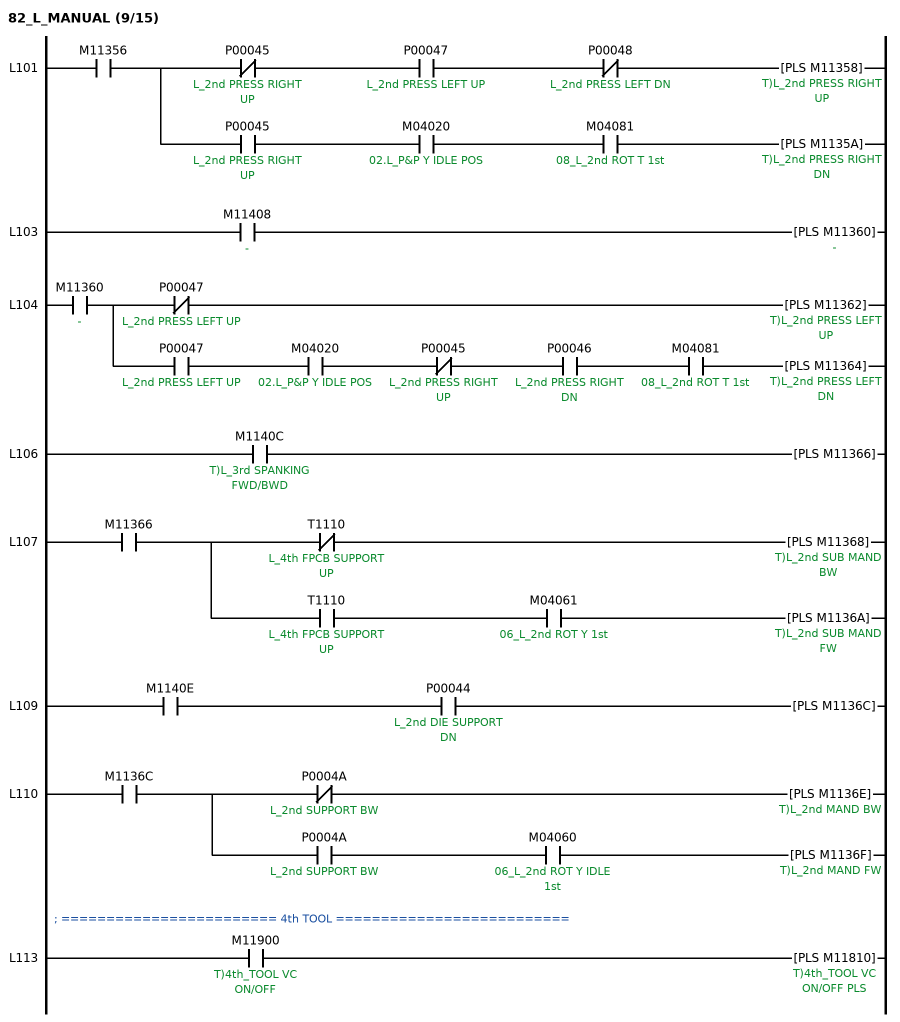
[picture p336: 82_L_MANUAL rungs L101-L113]
; L101
LOAD      M11356
MPUSH
AND NOT   P00045	// L_2nd PRESS RIGHT UP
AND       P00047	// L_2nd PRESS LEFT UP
AND NOT   P00048	// L_2nd PRESS LEFT DN
OUTP      M11358	// T)L_2nd PRESS RIGHT UP
MPOP
AND       P00045	// L_2nd PRESS RIGHT UP
AND       M04020	// 02.L_P&P Y IDLE POS
AND       M04081	// 08_L_2nd ROT T 1st
OUTP      M1135A	// T)L_2nd PRESS RIGHT DN
; L103
LOAD      M11408	// -
OUTP      M11360	// -
; L104
LOAD      M11360	// -
MPUSH
AND NOT   P00047	// L_2nd PRESS LEFT UP
OUTP      M11362	// T)L_2nd PRESS LEFT UP
MPOP
AND       P00047	// L_2nd PRESS LEFT UP
AND       M04020	// 02.L_P&P Y IDLE POS
AND NOT   P00045	// L_2nd PRESS RIGHT UP
AND       P00046	// L_2nd PRESS RIGHT DN
AND       M04081	// 08_L_2nd ROT T 1st
OUTP      M11364	// T)L_2nd PRESS LEFT DN
; L106
LOAD      M1140C	// T)L_3rd SPANKING FWD/BWD
OUTP      M11366
; L107
LOAD      M11366
MPUSH
AND NOT   T1110	// L_4th FPCB SUPPORT UP
OUTP      M11368	// T)L_2nd SUB MAND BW
MPOP
AND       T1110	// L_4th FPCB SUPPORT UP
AND       M04061	// 06_L_2nd ROT Y 1st
OUTP      M1136A	// T)L_2nd SUB MAND FW
; L109
LOAD      M1140E
AND       P00044	// L_2nd DIE SUPPORT DN
OUTP      M1136C
; L110
LOAD      M1136C
MPUSH
AND NOT   P0004A	// L_2nd SUPPORT BW
OUTP      M1136E	// T)L_2nd MAND BW
MPOP
AND       P0004A	// L_2nd SUPPORT BW
AND       M04060	// 06_L_2nd ROT Y IDLE 1st
OUTP      M1136F	// T)L_2nd MAND FW
// ======================== 4th TOOL ==========================
; L113
LOAD      M11900	// T)4th_TOOL VC ON/OFF
OUTP      M11810	// T)4th_TOOL VC ON/OFF PLS

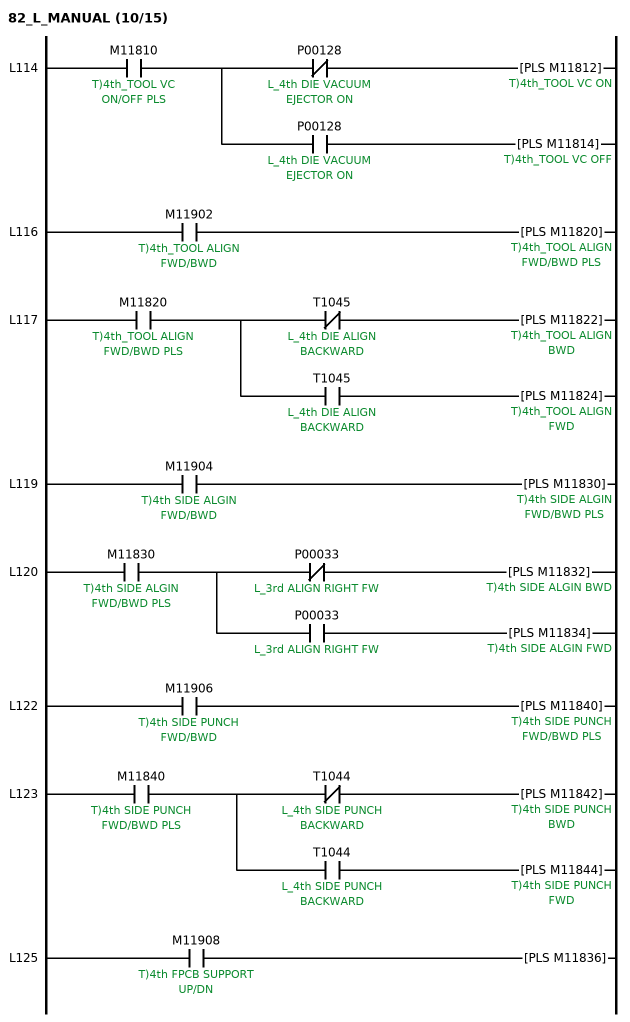
; L114
LOAD      M11810	// T)4th_TOOL VC ON/OFF PLS
MPUSH
AND NOT   P00128	// L_4th DIE VACUUM EJECTOR ON
OUTP      M11812	// T)4th_TOOL VC ON
MPOP
AND       P00128	// L_4th DIE VACUUM EJECTOR ON
OUTP      M11814	// T)4th_TOOL VC OFF
; L116
LOAD      M11902	// T)4th_TOOL ALIGN FWD/BWD
OUTP      M11820	// T)4th_TOOL ALIGN FWD/BWD PLS
; L117
LOAD      M11820	// T)4th_TOOL ALIGN FWD/BWD PLS
MPUSH
AND NOT   T1045	// L_4th DIE ALIGN BACKWARD
OUTP      M11822	// T)4th_TOOL ALIGN BWD
MPOP
AND       T1045	// L_4th DIE ALIGN BACKWARD
OUTP      M11824	// T)4th_TOOL ALIGN FWD
; L119
LOAD      M11904	// T)4th SIDE ALGIN FWD/BWD
OUTP      M11830	// T)4th SIDE ALGIN FWD/BWD PLS
; L120
LOAD      M11830	// T)4th SIDE ALGIN FWD/BWD PLS
MPUSH
AND NOT   P00033	// L_3rd ALIGN RIGHT FW
OUTP      M11832	// T)4th SIDE ALGIN BWD
MPOP
AND       P00033	// L_3rd ALIGN RIGHT FW
OUTP      M11834	// T)4th SIDE ALGIN FWD
; L122
LOAD      M11906	// T)4th SIDE PUNCH FWD/BWD
OUTP      M11840	// T)4th SIDE PUNCH FWD/BWD PLS
; L123
LOAD      M11840	// T)4th SIDE PUNCH FWD/BWD PLS
MPUSH
AND NOT   T1044	// L_4th SIDE PUNCH BACKWARD
OUTP      M11842	// T)4th SIDE PUNCH BWD
MPOP
AND       T1044	// L_4th SIDE PUNCH BACKWARD
OUTP      M11844	// T)4th SIDE PUNCH FWD
; L125
LOAD      M11908	// T)4th FPCB SUPPORT UP/DN
OUTP      M11836

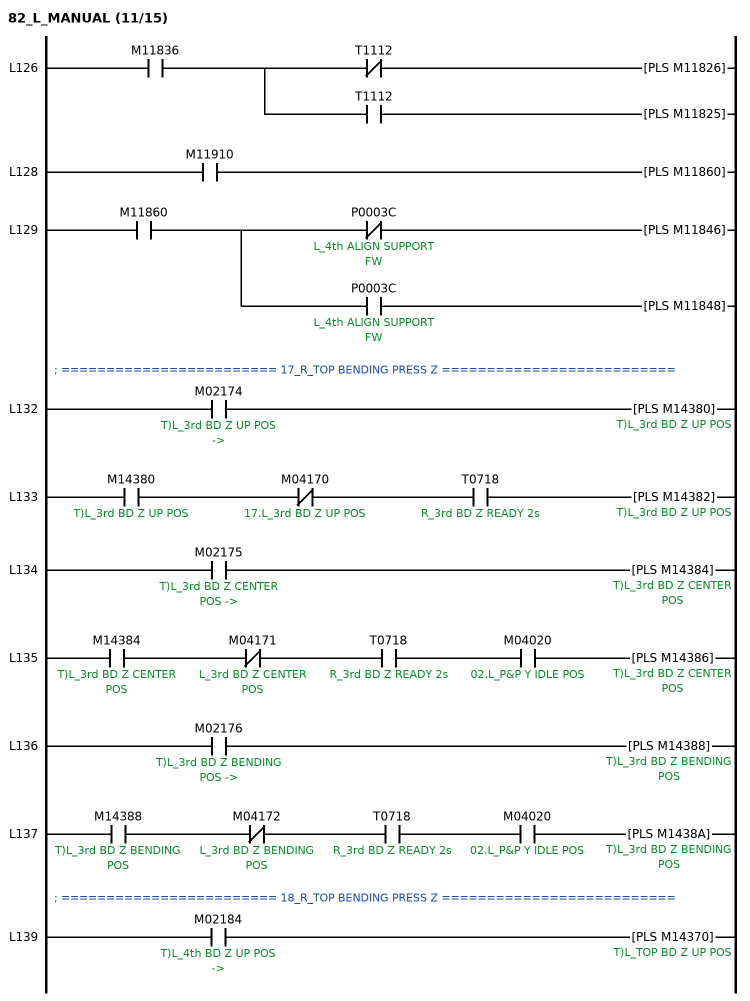
; L126
LOAD      M11836
MPUSH
AND NOT   T1112
OUTP      M11826
MPOP
AND       T1112
OUTP      M11825
; L128
LOAD      M11910
OUTP      M11860
; L129
LOAD      M11860
MPUSH
AND NOT   P0003C	// L_4th ALIGN SUPPORT FW
OUTP      M11846
MPOP
AND       P0003C	// L_4th ALIGN SUPPORT FW
OUTP      M11848
// ======================== 17_R_TOP BENDING PRESS Z ==========================
; L132
LOAD      M02174	// T)L_3rd BD Z UP POS ->
OUTP      M14380	// T)L_3rd BD Z UP POS
; L133
LOAD      M14380	// T)L_3rd BD Z UP POS
AND NOT   M04170	// 17.L_3rd BD Z UP POS
AND       T0718	// R_3rd BD Z READY 2s
OUTP      M14382	// T)L_3rd BD Z UP POS
; L134
LOAD      M02175	// T)L_3rd BD Z CENTER POS ->
OUTP      M14384	// T)L_3rd BD Z CENTER POS
; L135
LOAD      M14384	// T)L_3rd BD Z CENTER POS
AND NOT   M04171	// L_3rd BD Z CENTER POS
AND       T0718	// R_3rd BD Z READY 2s
AND       M04020	// 02.L_P&P Y IDLE POS
OUTP      M14386	// T)L_3rd BD Z CENTER POS
; L136
LOAD      M02176	// T)L_3rd BD Z BENDING POS ->
OUTP      M14388	// T)L_3rd BD Z BENDING POS
; L137
LOAD      M14388	// T)L_3rd BD Z BENDING POS
AND NOT   M04172	// L_3rd BD Z BENDING POS
AND       T0718	// R_3rd BD Z READY 2s
AND       M04020	// 02.L_P&P Y IDLE POS
OUTP      M1438A	// T)L_3rd BD Z BENDING POS
// ======================== 18_R_TOP BENDING PRESS Z ==========================
; L139
LOAD      M02184	// T)L_4th BD Z UP POS ->
OUTP      M14370	// T)L_TOP BD Z UP POS

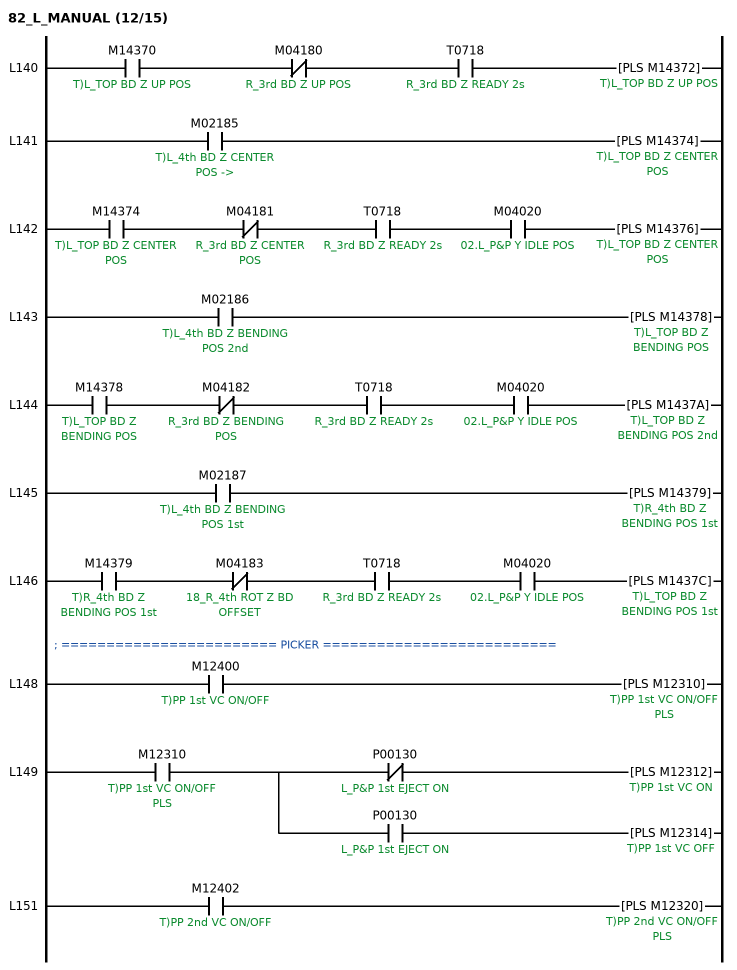
; L140
LOAD      M14370	// T)L_TOP BD Z UP POS
AND NOT   M04180	// R_3rd BD Z UP POS
AND       T0718	// R_3rd BD Z READY 2s
OUTP      M14372	// T)L_TOP BD Z UP POS
; L141
LOAD      M02185	// T)L_4th BD Z CENTER POS ->
OUTP      M14374	// T)L_TOP BD Z CENTER POS
; L142
LOAD      M14374	// T)L_TOP BD Z CENTER POS
AND NOT   M04181	// R_3rd BD Z CENTER POS
AND       T0718	// R_3rd BD Z READY 2s
AND       M04020	// 02.L_P&P Y IDLE POS
OUTP      M14376	// T)L_TOP BD Z CENTER POS
; L143
LOAD      M02186	// T)L_4th BD Z BENDING POS 2nd
OUTP      M14378	// T)L_TOP BD Z BENDING POS
; L144
LOAD      M14378	// T)L_TOP BD Z BENDING POS
AND NOT   M04182	// R_3rd BD Z BENDING POS
AND       T0718	// R_3rd BD Z READY 2s
AND       M04020	// 02.L_P&P Y IDLE POS
OUTP      M1437A	// T)L_TOP BD Z BENDING POS 2nd
; L145
LOAD      M02187	// T)L_4th BD Z BENDING POS 1st
OUTP      M14379	// T)R_4th BD Z BENDING POS 1st
; L146
LOAD      M14379	// T)R_4th BD Z BENDING POS 1st
AND NOT   M04183	// 18_R_4th ROT Z BD OFFSET
AND       T0718	// R_3rd BD Z READY 2s
AND       M04020	// 02.L_P&P Y IDLE POS
OUTP      M1437C	// T)L_TOP BD Z BENDING POS 1st
// ======================== PICKER ==========================
; L148
LOAD      M12400	// T)PP 1st VC ON/OFF
OUTP      M12310	// T)PP 1st VC ON/OFF PLS
; L149
LOAD      M12310	// T)PP 1st VC ON/OFF PLS
MPUSH
AND NOT   P00130	// L_P&P 1st EJECT ON
OUTP      M12312	// T)PP 1st VC ON
MPOP
AND       P00130	// L_P&P 1st EJECT ON
OUTP      M12314	// T)PP 1st VC OFF
; L151
LOAD      M12402	// T)PP 2nd VC ON/OFF
OUTP      M12320	// T)PP 2nd VC ON/OFF PLS

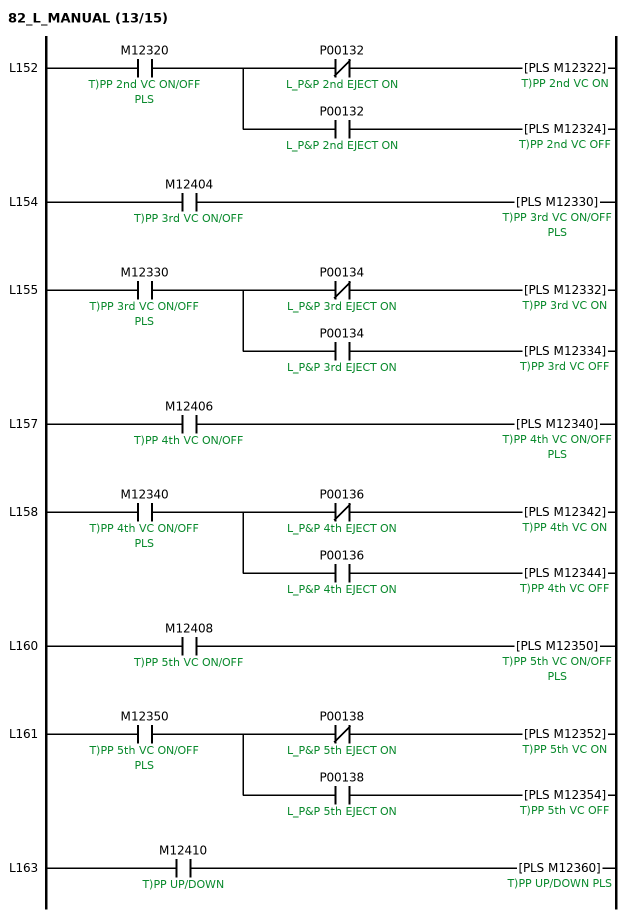
; L152
LOAD      M12320	// T)PP 2nd VC ON/OFF PLS
MPUSH
AND NOT   P00132	// L_P&P 2nd EJECT ON
OUTP      M12322	// T)PP 2nd VC ON
MPOP
AND       P00132	// L_P&P 2nd EJECT ON
OUTP      M12324	// T)PP 2nd VC OFF
; L154
LOAD      M12404	// T)PP 3rd VC ON/OFF
OUTP      M12330	// T)PP 3rd VC ON/OFF PLS
; L155
LOAD      M12330	// T)PP 3rd VC ON/OFF PLS
MPUSH
AND NOT   P00134	// L_P&P 3rd EJECT ON
OUTP      M12332	// T)PP 3rd VC ON
MPOP
AND       P00134	// L_P&P 3rd EJECT ON
OUTP      M12334	// T)PP 3rd VC OFF
; L157
LOAD      M12406	// T)PP 4th VC ON/OFF
OUTP      M12340	// T)PP 4th VC ON/OFF PLS
; L158
LOAD      M12340	// T)PP 4th VC ON/OFF PLS
MPUSH
AND NOT   P00136	// L_P&P 4th EJECT ON
OUTP      M12342	// T)PP 4th VC ON
MPOP
AND       P00136	// L_P&P 4th EJECT ON
OUTP      M12344	// T)PP 4th VC OFF
; L160
LOAD      M12408	// T)PP 5th VC ON/OFF
OUTP      M12350	// T)PP 5th VC ON/OFF PLS
; L161
LOAD      M12350	// T)PP 5th VC ON/OFF PLS
MPUSH
AND NOT   P00138	// L_P&P 5th EJECT ON
OUTP      M12352	// T)PP 5th VC ON
MPOP
AND       P00138	// L_P&P 5th EJECT ON
OUTP      M12354	// T)PP 5th VC OFF
; L163
LOAD      M12410	// T)PP UP/DOWN
OUTP      M12360	// T)PP UP/DOWN PLS

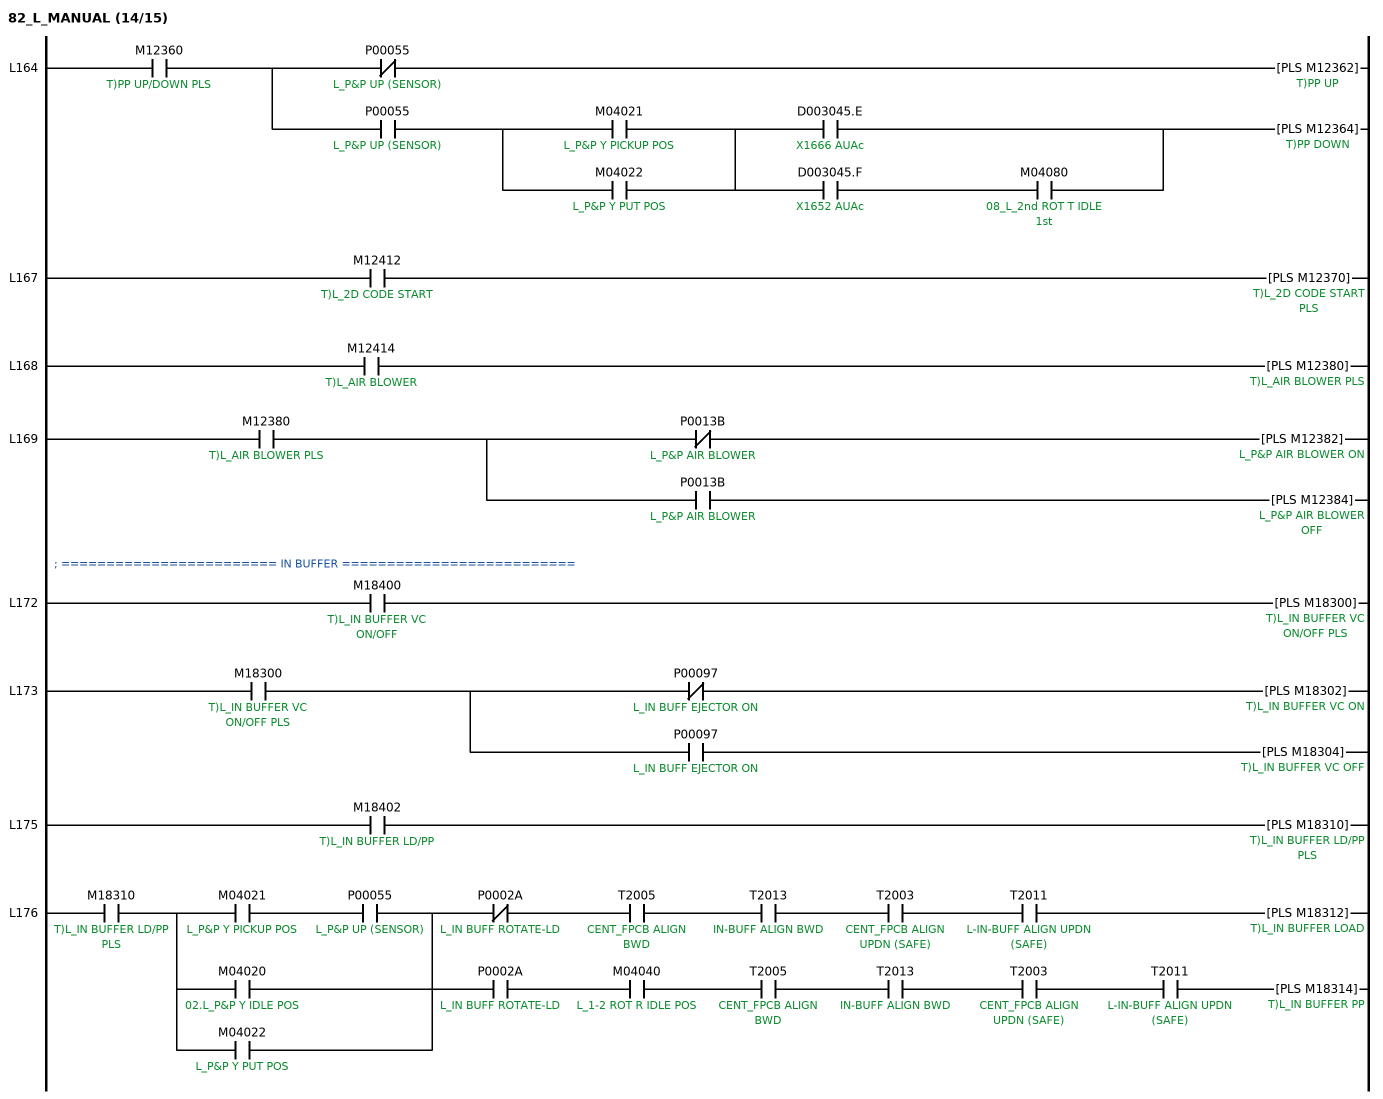
; L164
LOAD      M12360	// T)PP UP/DOWN PLS
MPUSH
AND NOT   P00055	// L_P&P UP (SENSOR)
OUTP      M12362	// T)PP UP
MPOP
AND       P00055	// L_P&P UP (SENSOR)
LOAD      M04021	// L_P&P Y PICKUP POS
OR        M04022	// L_P&P Y PUT POS
AND LOAD
LOAD      D003045.E	// X1666 AUAc
LOAD      D003045.F	// X1652 AUAc
AND       M04080	// 08_L_2nd ROT T IDLE 1st
OR LOAD
AND LOAD
OUTP      M12364	// T)PP DOWN
; L167
LOAD      M12412	// T)L_2D CODE START
OUTP      M12370	// T)L_2D CODE START PLS
; L168
LOAD      M12414	// T)L_AIR BLOWER
OUTP      M12380	// T)L_AIR BLOWER PLS
; L169
LOAD      M12380	// T)L_AIR BLOWER PLS
MPUSH
AND NOT   P0013B	// L_P&P AIR BLOWER
OUTP      M12382	// L_P&P AIR BLOWER ON
MPOP
AND       P0013B	// L_P&P AIR BLOWER
OUTP      M12384	// L_P&P AIR BLOWER OFF
// ======================== IN BUFFER ==========================
; L172
LOAD      M18400	// T)L_IN BUFFER VC ON/OFF
OUTP      M18300	// T)L_IN BUFFER VC ON/OFF PLS
; L173
LOAD      M18300	// T)L_IN BUFFER VC ON/OFF PLS
MPUSH
AND NOT   P00097	// L_IN BUFF EJECTOR ON
OUTP      M18302	// T)L_IN BUFFER VC ON
MPOP
AND       P00097	// L_IN BUFF EJECTOR ON
OUTP      M18304	// T)L_IN BUFFER VC OFF
; L175
LOAD      M18402	// T)L_IN BUFFER LD/PP
OUTP      M18310	// T)L_IN BUFFER LD/PP PLS
; L176
LOAD      M18310	// T)L_IN BUFFER LD/PP PLS
LOAD      M04021	// L_P&P Y PICKUP POS
AND       P00055	// L_P&P UP (SENSOR)
OR        M04020	// 02.L_P&P Y IDLE POS
OR        M04022	// L_P&P Y PUT POS
AND LOAD
MPUSH
AND NOT   P0002A	// L_IN BUFF ROTATE-LD
AND       T2005	// CENT_FPCB ALIGN BWD
AND       T2013	// IN-BUFF ALIGN BWD
AND       T2003	// CENT_FPCB ALIGN UPDN (SAFE)
AND       T2011	// L-IN-BUFF ALIGN UPDN (SAFE)
OUTP      M18312	// T)L_IN BUFFER LOAD
MPOP
AND       P0002A	// L_IN BUFF ROTATE-LD
AND       M04040	// L_1-2 ROT R IDLE POS
AND       T2005	// CENT_FPCB ALIGN BWD
AND       T2013	// IN-BUFF ALIGN BWD
AND       T2003	// CENT_FPCB ALIGN UPDN (SAFE)
AND       T2011	// L-IN-BUFF ALIGN UPDN (SAFE)
OUTP      M18314	// T)L_IN BUFFER PP

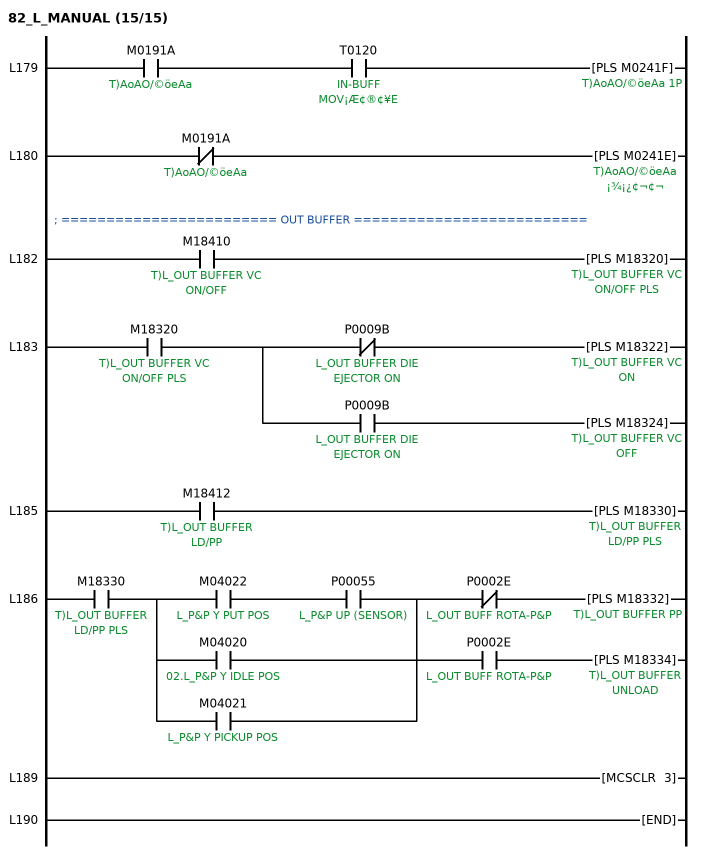
; L179
LOAD      M0191A	// T)AoAO/©öeAa
AND       T0120	// IN-BUFF MOV¡Æ¢®¢¥E
OUTP      M0241F	// T)AoAO/©öeAa 1P
; L180
LOAD NOT  M0191A	// T)AoAO/©öeAa
OUTP      M0241E	// T)AoAO/©öeAa ¡¾¡¿¢¬¢¬
// ======================== OUT BUFFER ==========================
; L182
LOAD      M18410	// T)L_OUT BUFFER VC ON/OFF
OUTP      M18320	// T)L_OUT BUFFER VC ON/OFF PLS
; L183
LOAD      M18320	// T)L_OUT BUFFER VC ON/OFF PLS
MPUSH
AND NOT   P0009B	// L_OUT BUFFER DIE EJECTOR ON
OUTP      M18322	// T)L_OUT BUFFER VC ON
MPOP
AND       P0009B	// L_OUT BUFFER DIE EJECTOR ON
OUTP      M18324	// T)L_OUT BUFFER VC OFF
; L185
LOAD      M18412	// T)L_OUT BUFFER LD/PP
OUTP      M18330	// T)L_OUT BUFFER LD/PP PLS
; L186
LOAD      M18330	// T)L_OUT BUFFER LD/PP PLS
LOAD      M04022	// L_P&P Y PUT POS
AND       P00055	// L_P&P UP (SENSOR)
OR        M04020	// 02.L_P&P Y IDLE POS
OR        M04021	// L_P&P Y PICKUP POS
AND LOAD
MPUSH
AND NOT   P0002E	// L_OUT BUFF ROTA-P&P
OUTP      M18332	// T)L_OUT BUFFER PP
MPOP
AND       P0002E	// L_OUT BUFF ROTA-P&P
OUTP      M18334	// T)L_OUT BUFFER UNLOAD
; L189
MCSCLR    3
; L190
END

PROGRAM 83_R_MANUAL (task: ¨ö¨¬A¥ì CA¡¤I¡¾¡¿¡¤¡Í)

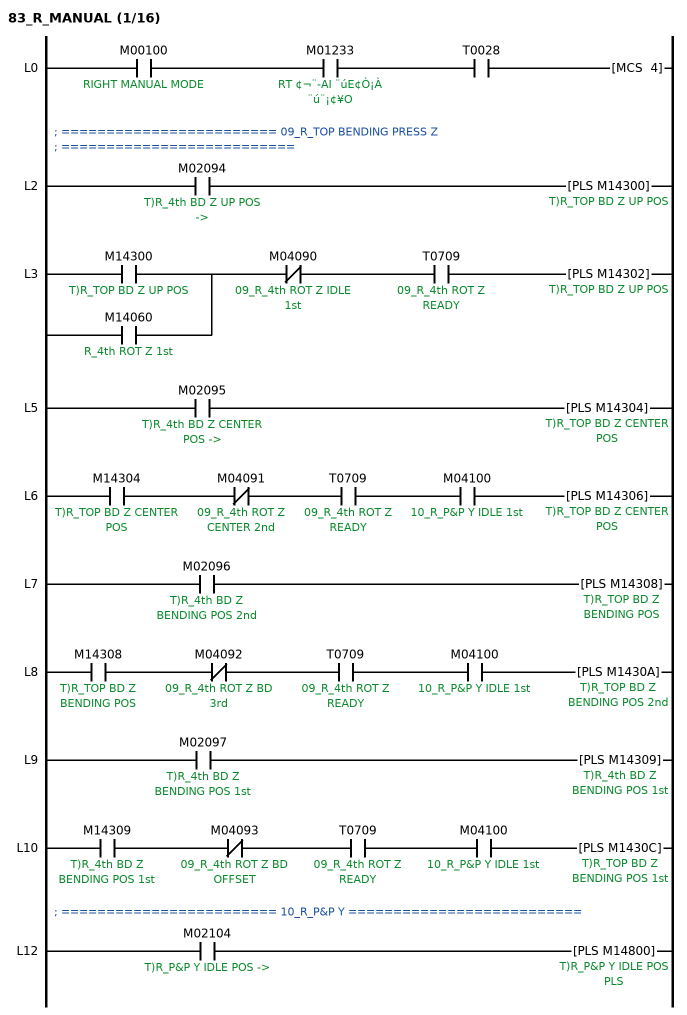
; L0
LOAD      M00100	// RIGHT MANUAL MODE
AND       M01233	// RT ¢¬¨­AI ¨úE¢Ò¡À ¨ú¨¡¢¥O
AND       T0028
MCS       4
// ======================== 09_R_TOP BENDING PRESS Z ==========================
; L2
LOAD      M02094	// T)R_4th BD Z UP POS ->
OUTP      M14300	// T)R_TOP BD Z UP POS
; L3
LOAD      M14300	// T)R_TOP BD Z UP POS
OR        M14060	// R_4th ROT Z 1st
AND NOT   M04090	// 09_R_4th ROT Z IDLE 1st
AND       T0709	// 09_R_4th ROT Z READY
OUTP      M14302	// T)R_TOP BD Z UP POS
; L5
LOAD      M02095	// T)R_4th BD Z CENTER POS ->
OUTP      M14304	// T)R_TOP BD Z CENTER POS
; L6
LOAD      M14304	// T)R_TOP BD Z CENTER POS
AND NOT   M04091	// 09_R_4th ROT Z CENTER 2nd
AND       T0709	// 09_R_4th ROT Z READY
AND       M04100	// 10_R_P&P Y IDLE 1st
OUTP      M14306	// T)R_TOP BD Z CENTER POS
; L7
LOAD      M02096	// T)R_4th BD Z BENDING POS 2nd
OUTP      M14308	// T)R_TOP BD Z BENDING POS
; L8
LOAD      M14308	// T)R_TOP BD Z BENDING POS
AND NOT   M04092	// 09_R_4th ROT Z BD 3rd
AND       T0709	// 09_R_4th ROT Z READY
AND       M04100	// 10_R_P&P Y IDLE 1st
OUTP      M1430A	// T)R_TOP BD Z BENDING POS 2nd
; L9
LOAD      M02097	// T)R_4th BD Z BENDING POS 1st
OUTP      M14309	// T)R_4th BD Z BENDING POS 1st
; L10
LOAD      M14309	// T)R_4th BD Z BENDING POS 1st
AND NOT   M04093	// 09_R_4th ROT Z BD OFFSET
AND       T0709	// 09_R_4th ROT Z READY
AND       M04100	// 10_R_P&P Y IDLE 1st
OUTP      M1430C	// T)R_TOP BD Z BENDING POS 1st
// ======================== 10_R_P&P Y ==========================
; L12
LOAD      M02104	// T)R_P&P Y IDLE POS ->
OUTP      M14800	// T)R_P&P Y IDLE POS PLS

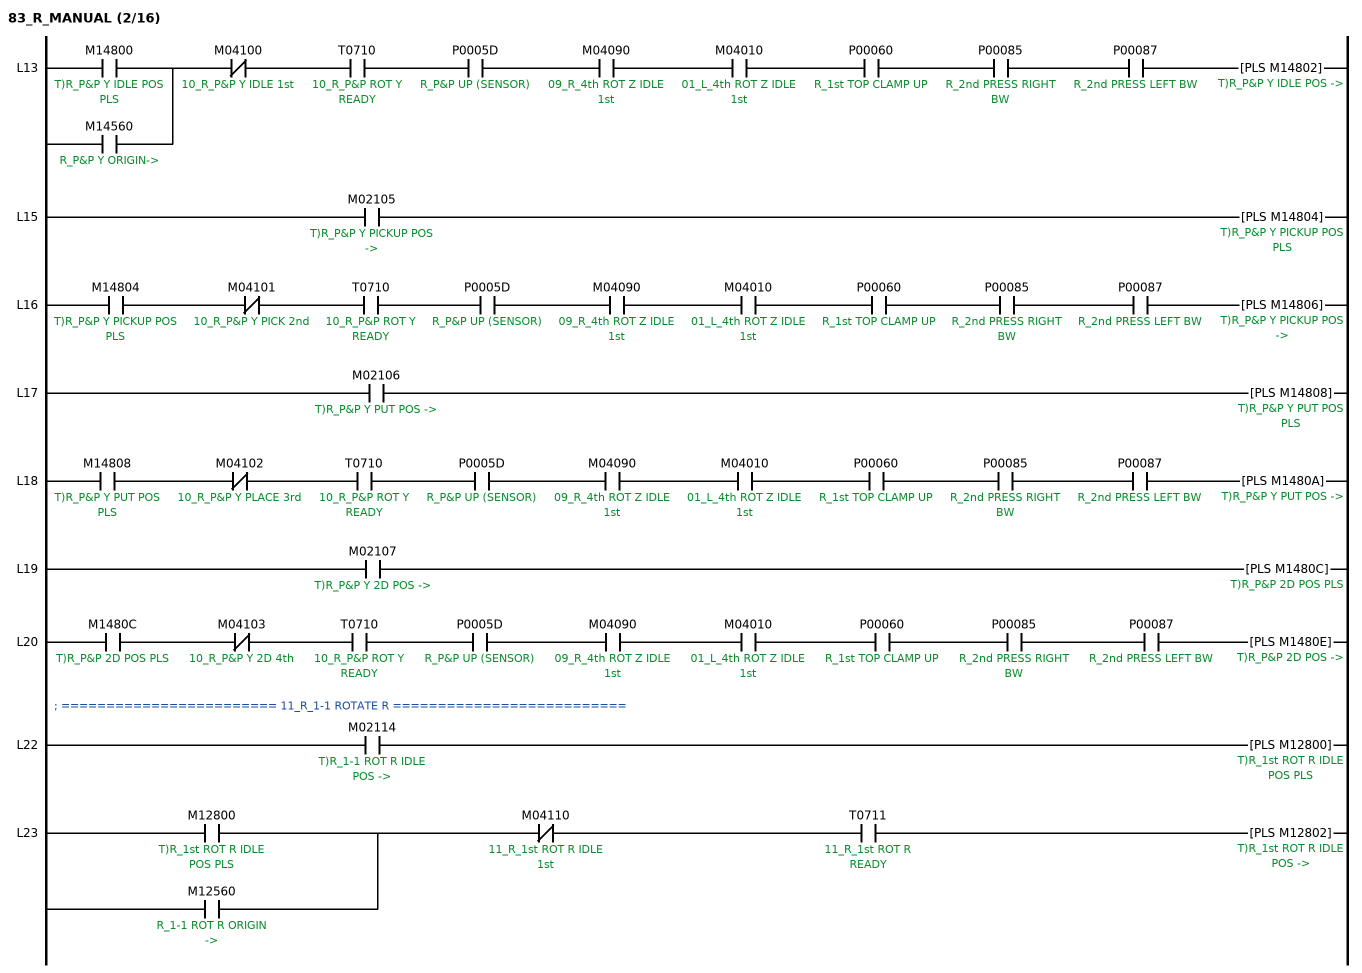
; L13
LOAD      M14800	// T)R_P&P Y IDLE POS PLS
OR        M14560	// R_P&P Y ORIGIN->
AND NOT   M04100	// 10_R_P&P Y IDLE 1st
AND       T0710	// 10_R_P&P ROT Y READY
AND       P0005D	// R_P&P UP (SENSOR)
AND       M04090	// 09_R_4th ROT Z IDLE 1st
AND       M04010	// 01_L_4th ROT Z IDLE 1st
AND       P00060	// R_1st TOP CLAMP UP
AND       P00085	// R_2nd PRESS RIGHT BW
AND       P00087	// R_2nd PRESS LEFT BW
OUTP      M14802	// T)R_P&P Y IDLE POS ->
; L15
LOAD      M02105	// T)R_P&P Y PICKUP POS ->
OUTP      M14804	// T)R_P&P Y PICKUP POS PLS
; L16
LOAD      M14804	// T)R_P&P Y PICKUP POS PLS
AND NOT   M04101	// 10_R_P&P Y PICK 2nd
AND       T0710	// 10_R_P&P ROT Y READY
AND       P0005D	// R_P&P UP (SENSOR)
AND       M04090	// 09_R_4th ROT Z IDLE 1st
AND       M04010	// 01_L_4th ROT Z IDLE 1st
AND       P00060	// R_1st TOP CLAMP UP
AND       P00085	// R_2nd PRESS RIGHT BW
AND       P00087	// R_2nd PRESS LEFT BW
OUTP      M14806	// T)R_P&P Y PICKUP POS ->
; L17
LOAD      M02106	// T)R_P&P Y PUT POS ->
OUTP      M14808	// T)R_P&P Y PUT POS PLS
; L18
LOAD      M14808	// T)R_P&P Y PUT POS PLS
AND NOT   M04102	// 10_R_P&P Y PLACE 3rd
AND       T0710	// 10_R_P&P ROT Y READY
AND       P0005D	// R_P&P UP (SENSOR)
AND       M04090	// 09_R_4th ROT Z IDLE 1st
AND       M04010	// 01_L_4th ROT Z IDLE 1st
AND       P00060	// R_1st TOP CLAMP UP
AND       P00085	// R_2nd PRESS RIGHT BW
AND       P00087	// R_2nd PRESS LEFT BW
OUTP      M1480A	// T)R_P&P Y PUT POS ->
; L19
LOAD      M02107	// T)R_P&P Y 2D POS ->
OUTP      M1480C	// T)R_P&P 2D POS PLS
; L20
LOAD      M1480C	// T)R_P&P 2D POS PLS
AND NOT   M04103	// 10_R_P&P Y 2D 4th
AND       T0710	// 10_R_P&P ROT Y READY
AND       P0005D	// R_P&P UP (SENSOR)
AND       M04090	// 09_R_4th ROT Z IDLE 1st
AND       M04010	// 01_L_4th ROT Z IDLE 1st
AND       P00060	// R_1st TOP CLAMP UP
AND       P00085	// R_2nd PRESS RIGHT BW
AND       P00087	// R_2nd PRESS LEFT BW
OUTP      M1480E	// T)R_P&P 2D POS ->
// ======================== 11_R_1-1 ROTATE R ==========================
; L22
LOAD      M02114	// T)R_1-1 ROT R IDLE POS ->
OUTP      M12800	// T)R_1st ROT R IDLE POS PLS
; L23
LOAD      M12800	// T)R_1st ROT R IDLE POS PLS
OR        M12560	// R_1-1 ROT R ORIGIN ->
AND NOT   M04110	// 11_R_1st ROT R IDLE 1st
AND       T0711	// 11_R_1st ROT R READY
OUTP      M12802	// T)R_1st ROT R IDLE POS ->

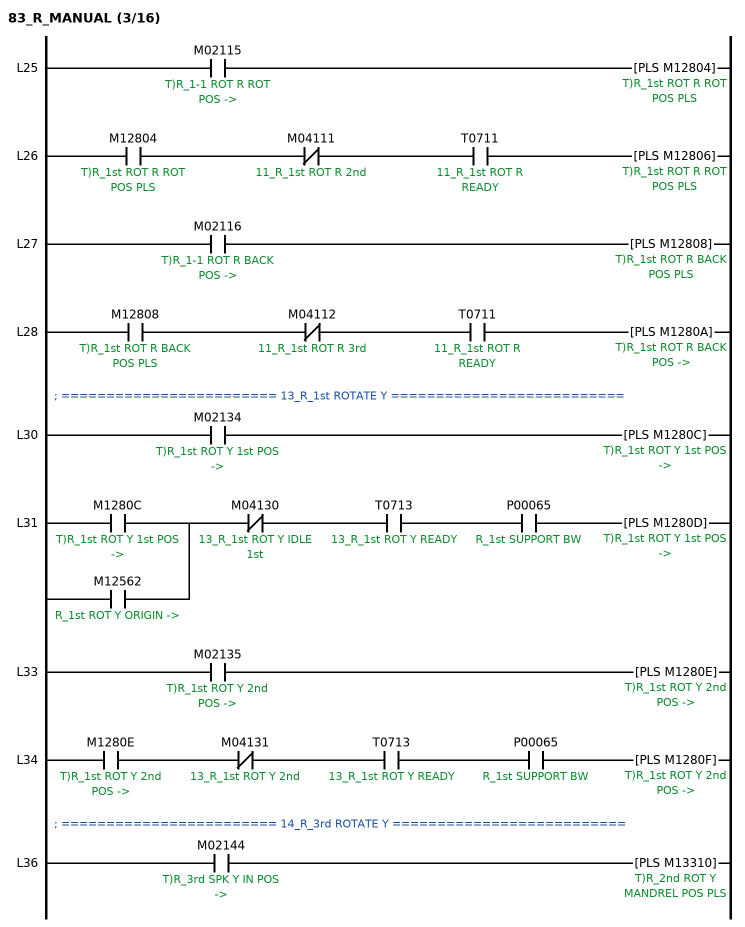
; L25
LOAD      M02115	// T)R_1-1 ROT R ROT POS ->
OUTP      M12804	// T)R_1st ROT R ROT POS PLS
; L26
LOAD      M12804	// T)R_1st ROT R ROT POS PLS
AND NOT   M04111	// 11_R_1st ROT R 2nd
AND       T0711	// 11_R_1st ROT R READY
OUTP      M12806	// T)R_1st ROT R ROT POS PLS
; L27
LOAD      M02116	// T)R_1-1 ROT R BACK POS ->
OUTP      M12808	// T)R_1st ROT R BACK POS PLS
; L28
LOAD      M12808	// T)R_1st ROT R BACK POS PLS
AND NOT   M04112	// 11_R_1st ROT R 3rd
AND       T0711	// 11_R_1st ROT R READY
OUTP      M1280A	// T)R_1st ROT R BACK POS ->
// ======================== 13_R_1st ROTATE Y ==========================
; L30
LOAD      M02134	// T)R_1st ROT Y 1st POS ->
OUTP      M1280C	// T)R_1st ROT Y 1st POS ->
; L31
LOAD      M1280C	// T)R_1st ROT Y 1st POS ->
OR        M12562	// R_1st ROT Y ORIGIN ->
AND NOT   M04130	// 13_R_1st ROT Y IDLE 1st
AND       T0713	// 13_R_1st ROT Y READY
AND       P00065	// R_1st SUPPORT BW
OUTP      M1280D	// T)R_1st ROT Y 1st POS ->
; L33
LOAD      M02135	// T)R_1st ROT Y 2nd POS ->
OUTP      M1280E	// T)R_1st ROT Y 2nd POS ->
; L34
LOAD      M1280E	// T)R_1st ROT Y 2nd POS ->
AND NOT   M04131	// 13_R_1st ROT Y 2nd
AND       T0713	// 13_R_1st ROT Y READY
AND       P00065	// R_1st SUPPORT BW
OUTP      M1280F	// T)R_1st ROT Y 2nd POS ->
// ======================== 14_R_3rd ROTATE Y ==========================
; L36
LOAD      M02144	// T)R_3rd SPK Y IN POS ->
OUTP      M13310	// T)R_2nd ROT Y MANDREL POS PLS

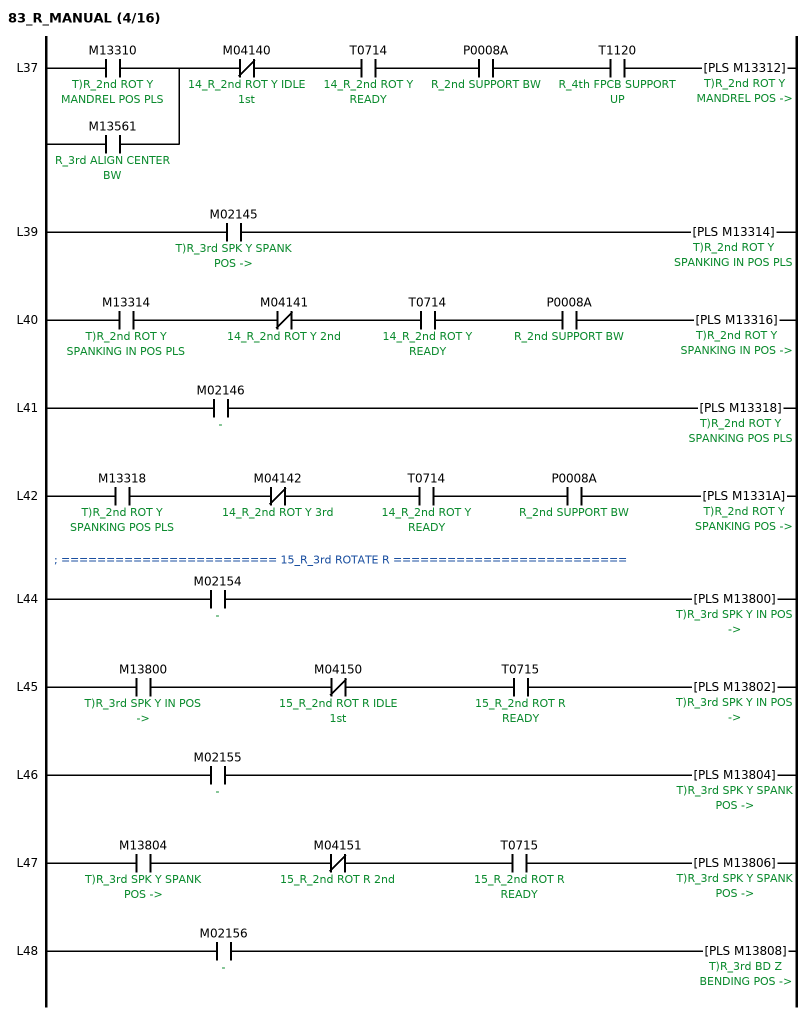
; L37
LOAD      M13310	// T)R_2nd ROT Y MANDREL POS PLS
OR        M13561	// R_3rd ALIGN CENTER BW
AND NOT   M04140	// 14_R_2nd ROT Y IDLE 1st
AND       T0714	// 14_R_2nd ROT Y READY
AND       P0008A	// R_2nd SUPPORT BW
AND       T1120	// R_4th FPCB SUPPORT UP
OUTP      M13312	// T)R_2nd ROT Y MANDREL POS ->
; L39
LOAD      M02145	// T)R_3rd SPK Y SPANK POS ->
OUTP      M13314	// T)R_2nd ROT Y SPANKING IN POS PLS
; L40
LOAD      M13314	// T)R_2nd ROT Y SPANKING IN POS PLS
AND NOT   M04141	// 14_R_2nd ROT Y 2nd
AND       T0714	// 14_R_2nd ROT Y READY
AND       P0008A	// R_2nd SUPPORT BW
OUTP      M13316	// T)R_2nd ROT Y SPANKING IN POS ->
; L41
LOAD      M02146	// -
OUTP      M13318	// T)R_2nd ROT Y SPANKING POS PLS
; L42
LOAD      M13318	// T)R_2nd ROT Y SPANKING POS PLS
AND NOT   M04142	// 14_R_2nd ROT Y 3rd
AND       T0714	// 14_R_2nd ROT Y READY
AND       P0008A	// R_2nd SUPPORT BW
OUTP      M1331A	// T)R_2nd ROT Y SPANKING POS ->
// ======================== 15_R_3rd ROTATE R ==========================
; L44
LOAD      M02154	// -
OUTP      M13800	// T)R_3rd SPK Y IN POS ->
; L45
LOAD      M13800	// T)R_3rd SPK Y IN POS ->
AND NOT   M04150	// 15_R_2nd ROT R IDLE 1st
AND       T0715	// 15_R_2nd ROT R READY
OUTP      M13802	// T)R_3rd SPK Y IN POS ->
; L46
LOAD      M02155	// -
OUTP      M13804	// T)R_3rd SPK Y SPANK POS ->
; L47
LOAD      M13804	// T)R_3rd SPK Y SPANK POS ->
AND NOT   M04151	// 15_R_2nd ROT R 2nd
AND       T0715	// 15_R_2nd ROT R READY
OUTP      M13806	// T)R_3rd SPK Y SPANK POS ->
; L48
LOAD      M02156	// -
OUTP      M13808	// T)R_3rd BD Z BENDING POS ->

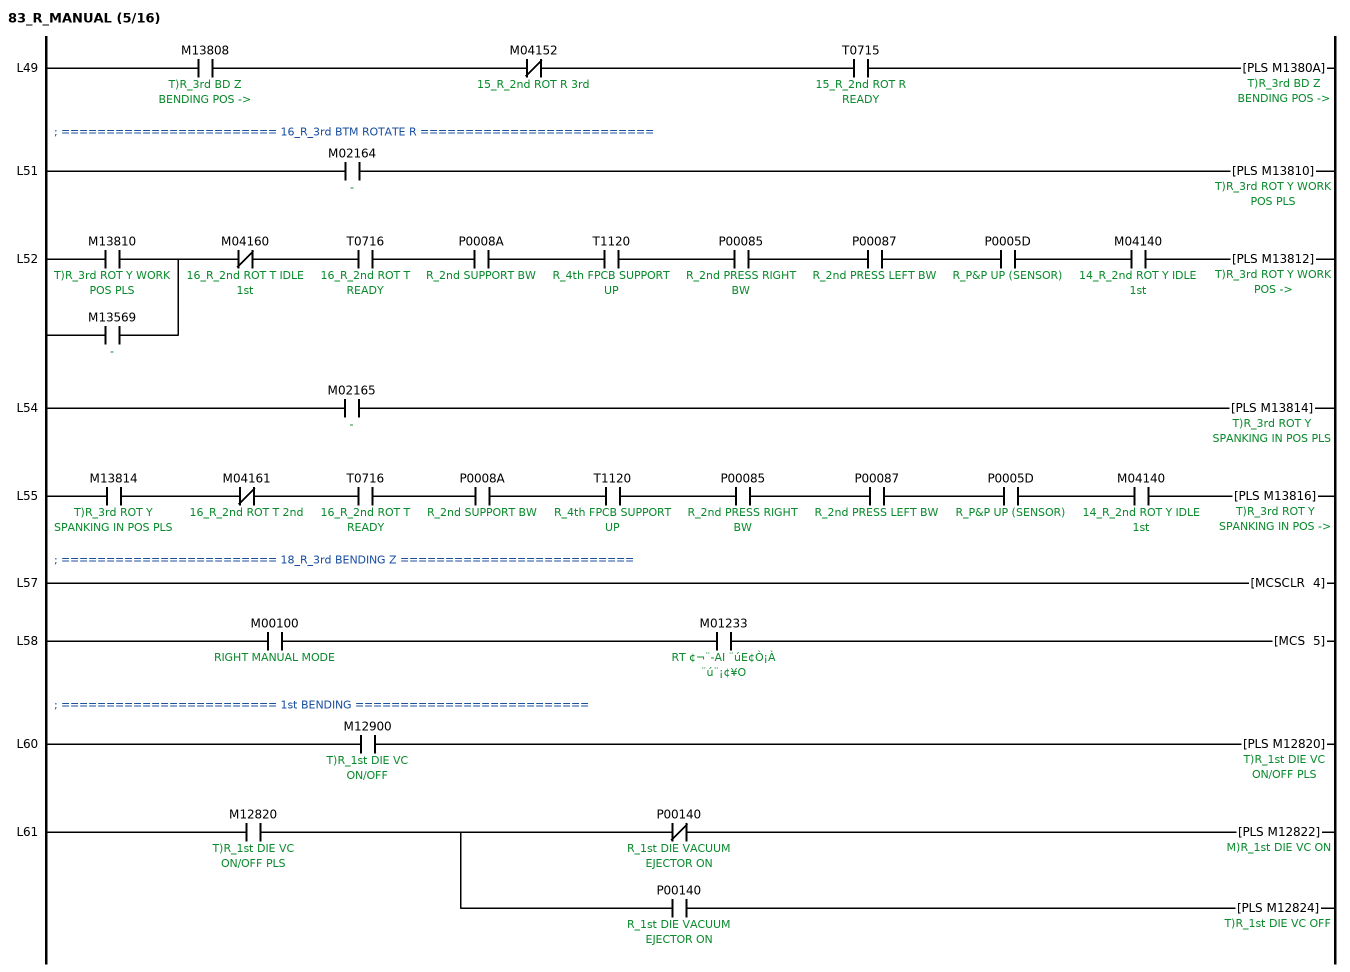
; L49
LOAD      M13808	// T)R_3rd BD Z BENDING POS ->
AND NOT   M04152	// 15_R_2nd ROT R 3rd
AND       T0715	// 15_R_2nd ROT R READY
OUTP      M1380A	// T)R_3rd BD Z BENDING POS ->
// ======================== 16_R_3rd BTM ROTATE R ==========================
; L51
LOAD      M02164	// -
OUTP      M13810	// T)R_3rd ROT Y WORK POS PLS
; L52
LOAD      M13810	// T)R_3rd ROT Y WORK POS PLS
OR        M13569	// -
AND NOT   M04160	// 16_R_2nd ROT T IDLE 1st
AND       T0716	// 16_R_2nd ROT T READY
AND       P0008A	// R_2nd SUPPORT BW
AND       T1120	// R_4th FPCB SUPPORT UP
AND       P00085	// R_2nd PRESS RIGHT BW
AND       P00087	// R_2nd PRESS LEFT BW
AND       P0005D	// R_P&P UP (SENSOR)
AND       M04140	// 14_R_2nd ROT Y IDLE 1st
OUTP      M13812	// T)R_3rd ROT Y WORK POS ->
; L54
LOAD      M02165	// -
OUTP      M13814	// T)R_3rd ROT Y SPANKING IN POS PLS
; L55
LOAD      M13814	// T)R_3rd ROT Y SPANKING IN POS PLS
AND NOT   M04161	// 16_R_2nd ROT T 2nd
AND       T0716	// 16_R_2nd ROT T READY
AND       P0008A	// R_2nd SUPPORT BW
AND       T1120	// R_4th FPCB SUPPORT UP
AND       P00085	// R_2nd PRESS RIGHT BW
AND       P00087	// R_2nd PRESS LEFT BW
AND       P0005D	// R_P&P UP (SENSOR)
AND       M04140	// 14_R_2nd ROT Y IDLE 1st
OUTP      M13816	// T)R_3rd ROT Y SPANKING IN POS ->
// ======================== 18_R_3rd BENDING Z ==========================
; L57
MCSCLR    4
; L58
LOAD      M00100	// RIGHT MANUAL MODE
AND       M01233	// RT ¢¬¨­AI ¨úE¢Ò¡À ¨ú¨¡¢¥O
MCS       5
// ======================== 1st BENDING ==========================
; L60
LOAD      M12900	// T)R_1st DIE VC ON/OFF
OUTP      M12820	// T)R_1st DIE VC ON/OFF PLS
; L61
LOAD      M12820	// T)R_1st DIE VC ON/OFF PLS
MPUSH
AND NOT   P00140	// R_1st DIE VACUUM EJECTOR ON
OUTP      M12822	// M)R_1st DIE VC ON
MPOP
AND       P00140	// R_1st DIE VACUUM EJECTOR ON
OUTP      M12824	// T)R_1st DIE VC OFF

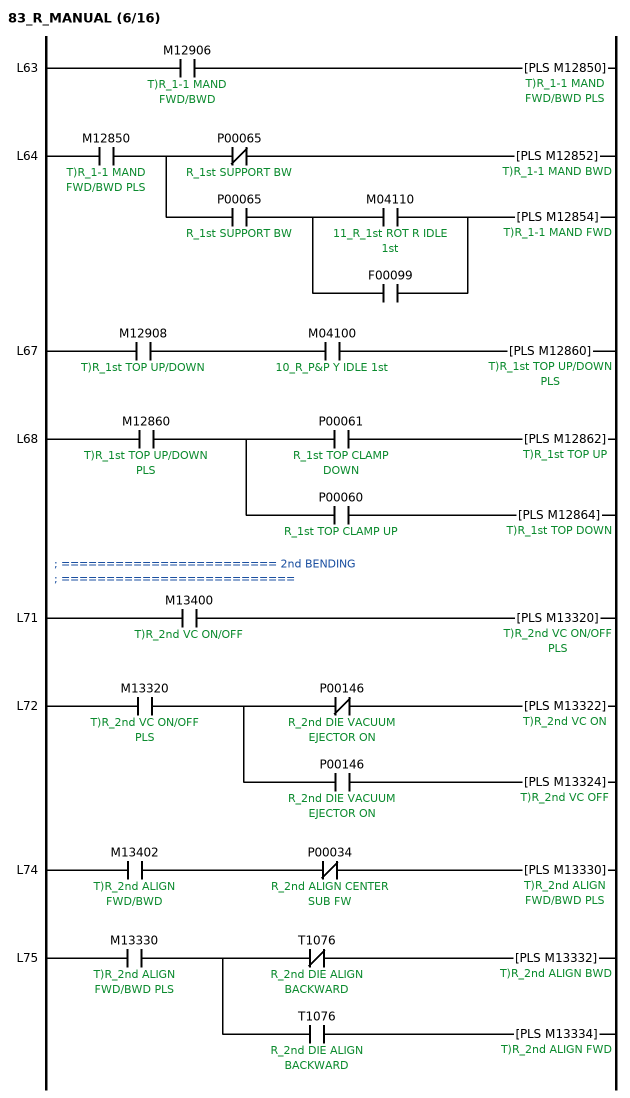
; L63
LOAD      M12906	// T)R_1-1 MAND FWD/BWD
OUTP      M12850	// T)R_1-1 MAND FWD/BWD PLS
; L64
LOAD      M12850	// T)R_1-1 MAND FWD/BWD PLS
MPUSH
AND NOT   P00065	// R_1st SUPPORT BW
OUTP      M12852	// T)R_1-1 MAND BWD
MPOP
AND       P00065	// R_1st SUPPORT BW
LOAD      M04110	// 11_R_1st ROT R IDLE 1st
OR        F00099
AND LOAD
OUTP      M12854	// T)R_1-1 MAND FWD
; L67
LOAD      M12908	// T)R_1st TOP UP/DOWN
AND       M04100	// 10_R_P&P Y IDLE 1st
OUTP      M12860	// T)R_1st TOP UP/DOWN PLS
; L68
LOAD      M12860	// T)R_1st TOP UP/DOWN PLS
MPUSH
AND       P00061	// R_1st TOP CLAMP DOWN
OUTP      M12862	// T)R_1st TOP UP
MPOP
AND       P00060	// R_1st TOP CLAMP UP
OUTP      M12864	// T)R_1st TOP DOWN
// ======================== 2nd BENDING ==========================
; L71
LOAD      M13400	// T)R_2nd VC ON/OFF
OUTP      M13320	// T)R_2nd VC ON/OFF PLS
; L72
LOAD      M13320	// T)R_2nd VC ON/OFF PLS
MPUSH
AND NOT   P00146	// R_2nd DIE VACUUM EJECTOR ON
OUTP      M13322	// T)R_2nd VC ON
MPOP
AND       P00146	// R_2nd DIE VACUUM EJECTOR ON
OUTP      M13324	// T)R_2nd VC OFF
; L74
LOAD      M13402	// T)R_2nd ALIGN FWD/BWD
AND NOT   P00034	// R_2nd ALIGN CENTER SUB FW
OUTP      M13330	// T)R_2nd ALIGN FWD/BWD PLS
; L75
LOAD      M13330	// T)R_2nd ALIGN FWD/BWD PLS
MPUSH
AND NOT   T1076	// R_2nd DIE ALIGN BACKWARD
OUTP      M13332	// T)R_2nd ALIGN BWD
MPOP
AND       T1076	// R_2nd DIE ALIGN BACKWARD
OUTP      M13334	// T)R_2nd ALIGN FWD

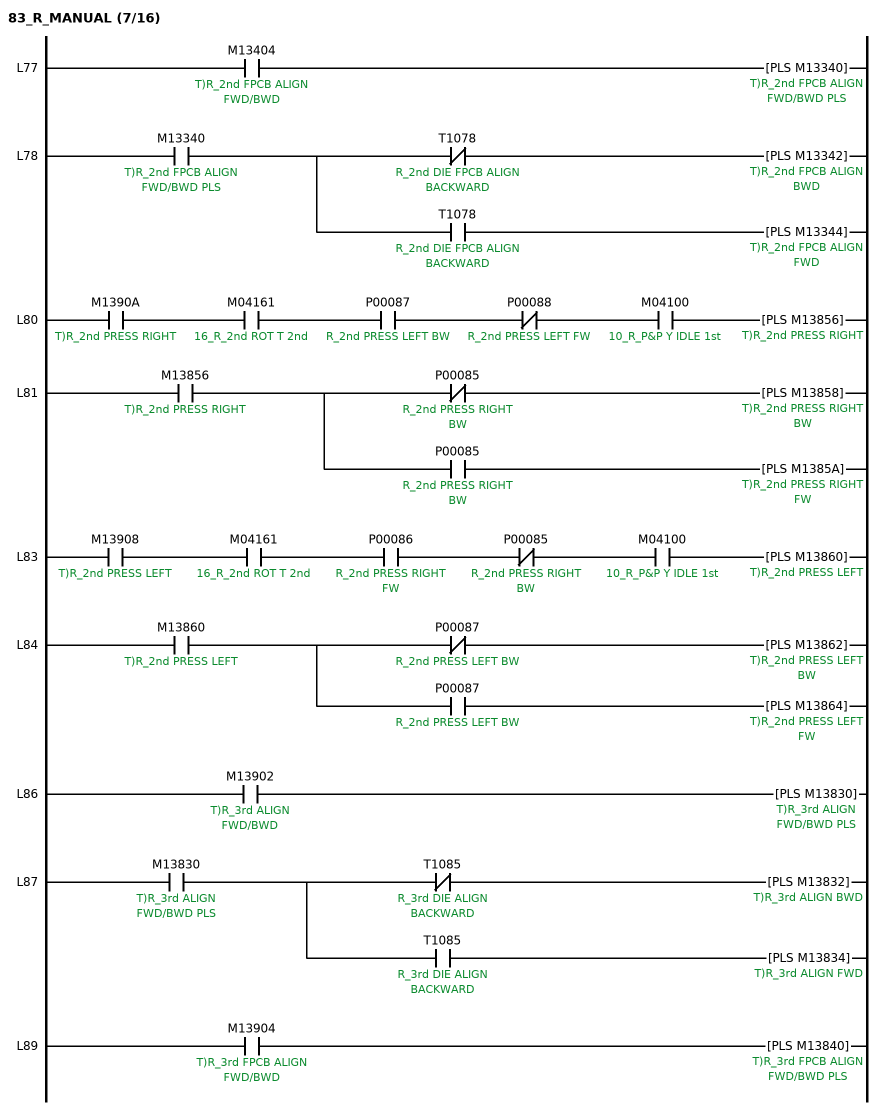
; L77
LOAD      M13404	// T)R_2nd FPCB ALIGN FWD/BWD
OUTP      M13340	// T)R_2nd FPCB ALIGN FWD/BWD PLS
; L78
LOAD      M13340	// T)R_2nd FPCB ALIGN FWD/BWD PLS
MPUSH
AND NOT   T1078	// R_2nd DIE FPCB ALIGN BACKWARD
OUTP      M13342	// T)R_2nd FPCB ALIGN BWD
MPOP
AND       T1078	// R_2nd DIE FPCB ALIGN BACKWARD
OUTP      M13344	// T)R_2nd FPCB ALIGN FWD
; L80
LOAD      M1390A	// T)R_2nd PRESS RIGHT
AND       M04161	// 16_R_2nd ROT T 2nd
AND       P00087	// R_2nd PRESS LEFT BW
AND NOT   P00088	// R_2nd PRESS LEFT FW
AND       M04100	// 10_R_P&P Y IDLE 1st
OUTP      M13856	// T)R_2nd PRESS RIGHT
; L81
LOAD      M13856	// T)R_2nd PRESS RIGHT
MPUSH
AND NOT   P00085	// R_2nd PRESS RIGHT BW
OUTP      M13858	// T)R_2nd PRESS RIGHT BW
MPOP
AND       P00085	// R_2nd PRESS RIGHT BW
OUTP      M1385A	// T)R_2nd PRESS RIGHT FW
; L83
LOAD      M13908	// T)R_2nd PRESS LEFT
AND       M04161	// 16_R_2nd ROT T 2nd
AND       P00086	// R_2nd PRESS RIGHT FW
AND NOT   P00085	// R_2nd PRESS RIGHT BW
AND       M04100	// 10_R_P&P Y IDLE 1st
OUTP      M13860	// T)R_2nd PRESS LEFT
; L84
LOAD      M13860	// T)R_2nd PRESS LEFT
MPUSH
AND NOT   P00087	// R_2nd PRESS LEFT BW
OUTP      M13862	// T)R_2nd PRESS LEFT BW
MPOP
AND       P00087	// R_2nd PRESS LEFT BW
OUTP      M13864	// T)R_2nd PRESS LEFT FW
; L86
LOAD      M13902	// T)R_3rd ALIGN FWD/BWD
OUTP      M13830	// T)R_3rd ALIGN FWD/BWD PLS
; L87
LOAD      M13830	// T)R_3rd ALIGN FWD/BWD PLS
MPUSH
AND NOT   T1085	// R_3rd DIE ALIGN BACKWARD
OUTP      M13832	// T)R_3rd ALIGN BWD
MPOP
AND       T1085	// R_3rd DIE ALIGN BACKWARD
OUTP      M13834	// T)R_3rd ALIGN FWD
; L89
LOAD      M13904	// T)R_3rd FPCB ALIGN FWD/BWD
OUTP      M13840	// T)R_3rd FPCB ALIGN FWD/BWD PLS

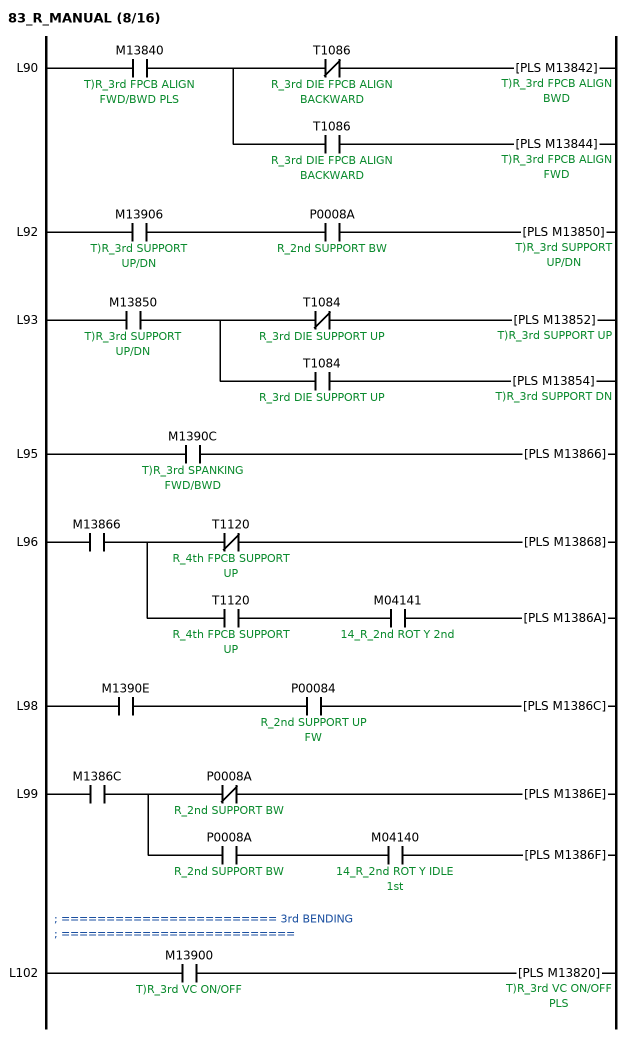
; L90
LOAD      M13840	// T)R_3rd FPCB ALIGN FWD/BWD PLS
MPUSH
AND NOT   T1086	// R_3rd DIE FPCB ALIGN BACKWARD
OUTP      M13842	// T)R_3rd FPCB ALIGN BWD
MPOP
AND       T1086	// R_3rd DIE FPCB ALIGN BACKWARD
OUTP      M13844	// T)R_3rd FPCB ALIGN FWD
; L92
LOAD      M13906	// T)R_3rd SUPPORT UP/DN
AND       P0008A	// R_2nd SUPPORT BW
OUTP      M13850	// T)R_3rd SUPPORT UP/DN
; L93
LOAD      M13850	// T)R_3rd SUPPORT UP/DN
MPUSH
AND NOT   T1084	// R_3rd DIE SUPPORT UP
OUTP      M13852	// T)R_3rd SUPPORT UP
MPOP
AND       T1084	// R_3rd DIE SUPPORT UP
OUTP      M13854	// T)R_3rd SUPPORT DN
; L95
LOAD      M1390C	// T)R_3rd SPANKING FWD/BWD
OUTP      M13866
; L96
LOAD      M13866
MPUSH
AND NOT   T1120	// R_4th FPCB SUPPORT UP
OUTP      M13868
MPOP
AND       T1120	// R_4th FPCB SUPPORT UP
AND       M04141	// 14_R_2nd ROT Y 2nd
OUTP      M1386A
; L98
LOAD      M1390E
AND       P00084	// R_2nd SUPPORT UP FW
OUTP      M1386C
; L99
LOAD      M1386C
MPUSH
AND NOT   P0008A	// R_2nd SUPPORT BW
OUTP      M1386E
MPOP
AND       P0008A	// R_2nd SUPPORT BW
AND       M04140	// 14_R_2nd ROT Y IDLE 1st
OUTP      M1386F
// ======================== 3rd BENDING ==========================
; L102
LOAD      M13900	// T)R_3rd VC ON/OFF
OUTP      M13820	// T)R_3rd VC ON/OFF PLS

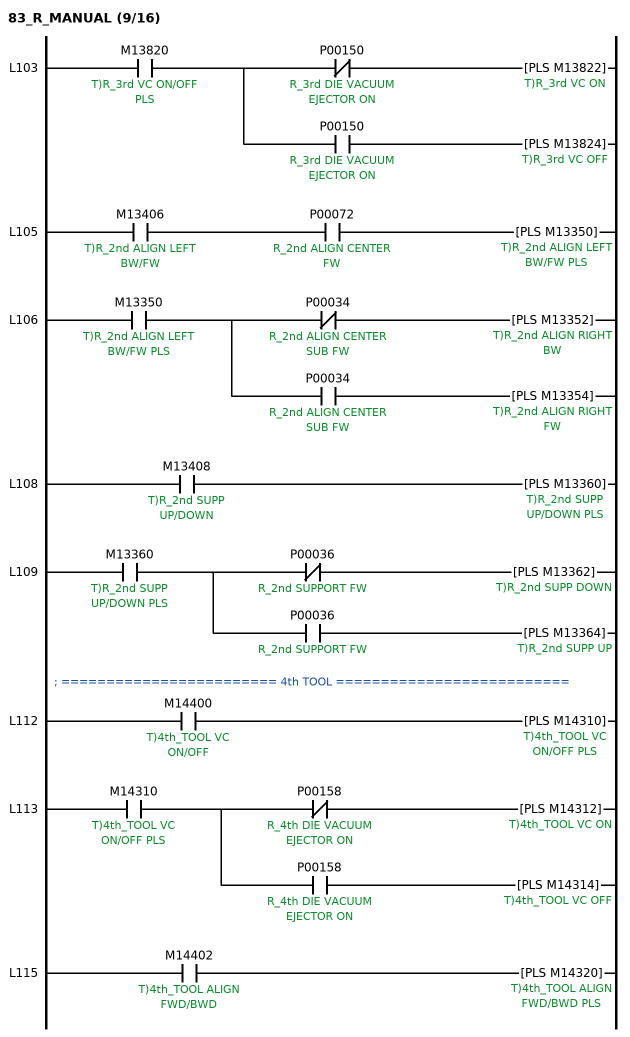
; L103
LOAD      M13820	// T)R_3rd VC ON/OFF PLS
MPUSH
AND NOT   P00150	// R_3rd DIE VACUUM EJECTOR ON
OUTP      M13822	// T)R_3rd VC ON
MPOP
AND       P00150	// R_3rd DIE VACUUM EJECTOR ON
OUTP      M13824	// T)R_3rd VC OFF
; L105
LOAD      M13406	// T)R_2nd ALIGN LEFT BW/FW
AND       P00072	// R_2nd ALIGN CENTER FW
OUTP      M13350	// T)R_2nd ALIGN LEFT BW/FW PLS
; L106
LOAD      M13350	// T)R_2nd ALIGN LEFT BW/FW PLS
MPUSH
AND NOT   P00034	// R_2nd ALIGN CENTER SUB FW
OUTP      M13352	// T)R_2nd ALIGN RIGHT BW
MPOP
AND       P00034	// R_2nd ALIGN CENTER SUB FW
OUTP      M13354	// T)R_2nd ALIGN RIGHT FW
; L108
LOAD      M13408	// T)R_2nd SUPP UP/DOWN
OUTP      M13360	// T)R_2nd SUPP UP/DOWN PLS
; L109
LOAD      M13360	// T)R_2nd SUPP UP/DOWN PLS
MPUSH
AND NOT   P00036	// R_2nd SUPPORT FW
OUTP      M13362	// T)R_2nd SUPP DOWN
MPOP
AND       P00036	// R_2nd SUPPORT FW
OUTP      M13364	// T)R_2nd SUPP UP
// ======================== 4th TOOL ==========================
; L112
LOAD      M14400	// T)4th_TOOL VC ON/OFF
OUTP      M14310	// T)4th_TOOL VC ON/OFF PLS
; L113
LOAD      M14310	// T)4th_TOOL VC ON/OFF PLS
MPUSH
AND NOT   P00158	// R_4th DIE VACUUM EJECTOR ON
OUTP      M14312	// T)4th_TOOL VC ON
MPOP
AND       P00158	// R_4th DIE VACUUM EJECTOR ON
OUTP      M14314	// T)4th_TOOL VC OFF
; L115
LOAD      M14402	// T)4th_TOOL ALIGN FWD/BWD
OUTP      M14320	// T)4th_TOOL ALIGN FWD/BWD PLS

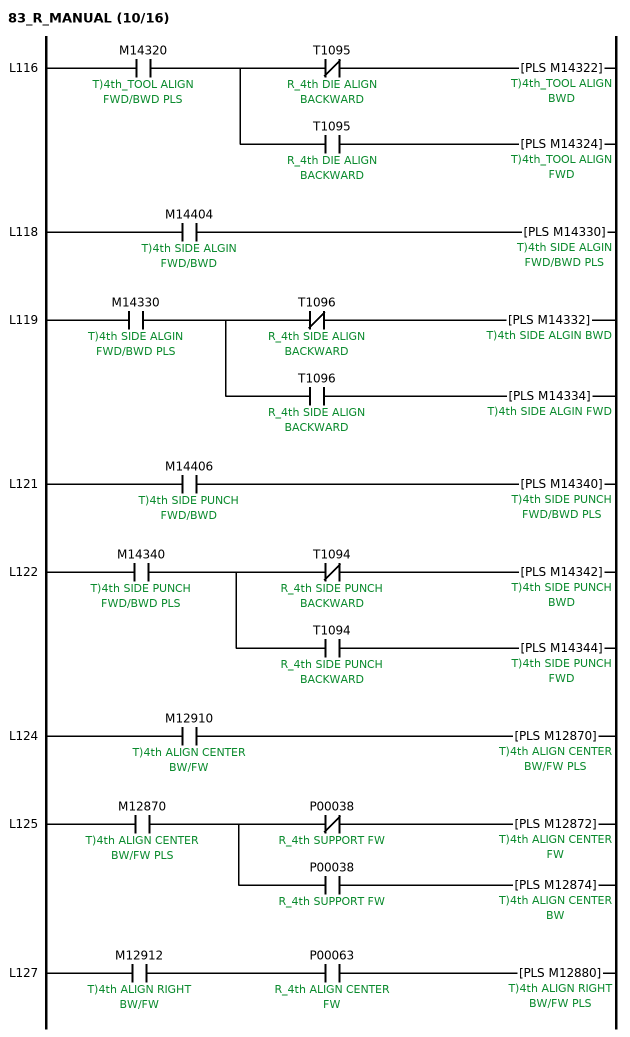
; L116
LOAD      M14320	// T)4th_TOOL ALIGN FWD/BWD PLS
MPUSH
AND NOT   T1095	// R_4th DIE ALIGN BACKWARD
OUTP      M14322	// T)4th_TOOL ALIGN BWD
MPOP
AND       T1095	// R_4th DIE ALIGN BACKWARD
OUTP      M14324	// T)4th_TOOL ALIGN FWD
; L118
LOAD      M14404	// T)4th SIDE ALGIN FWD/BWD
OUTP      M14330	// T)4th SIDE ALGIN FWD/BWD PLS
; L119
LOAD      M14330	// T)4th SIDE ALGIN FWD/BWD PLS
MPUSH
AND NOT   T1096	// R_4th SIDE ALIGN BACKWARD
OUTP      M14332	// T)4th SIDE ALGIN BWD
MPOP
AND       T1096	// R_4th SIDE ALIGN BACKWARD
OUTP      M14334	// T)4th SIDE ALGIN FWD
; L121
LOAD      M14406	// T)4th SIDE PUNCH FWD/BWD
OUTP      M14340	// T)4th SIDE PUNCH FWD/BWD PLS
; L122
LOAD      M14340	// T)4th SIDE PUNCH FWD/BWD PLS
MPUSH
AND NOT   T1094	// R_4th SIDE PUNCH BACKWARD
OUTP      M14342	// T)4th SIDE PUNCH BWD
MPOP
AND       T1094	// R_4th SIDE PUNCH BACKWARD
OUTP      M14344	// T)4th SIDE PUNCH FWD
; L124
LOAD      M12910	// T)4th ALIGN CENTER BW/FW
OUTP      M12870	// T)4th ALIGN CENTER BW/FW PLS
; L125
LOAD      M12870	// T)4th ALIGN CENTER BW/FW PLS
MPUSH
AND NOT   P00038	// R_4th SUPPORT FW
OUTP      M12872	// T)4th ALIGN CENTER FW
MPOP
AND       P00038	// R_4th SUPPORT FW
OUTP      M12874	// T)4th ALIGN CENTER BW
; L127
LOAD      M12912	// T)4th ALIGN RIGHT BW/FW
AND       P00063	// R_4th ALIGN CENTER FW
OUTP      M12880	// T)4th ALIGN RIGHT BW/FW PLS

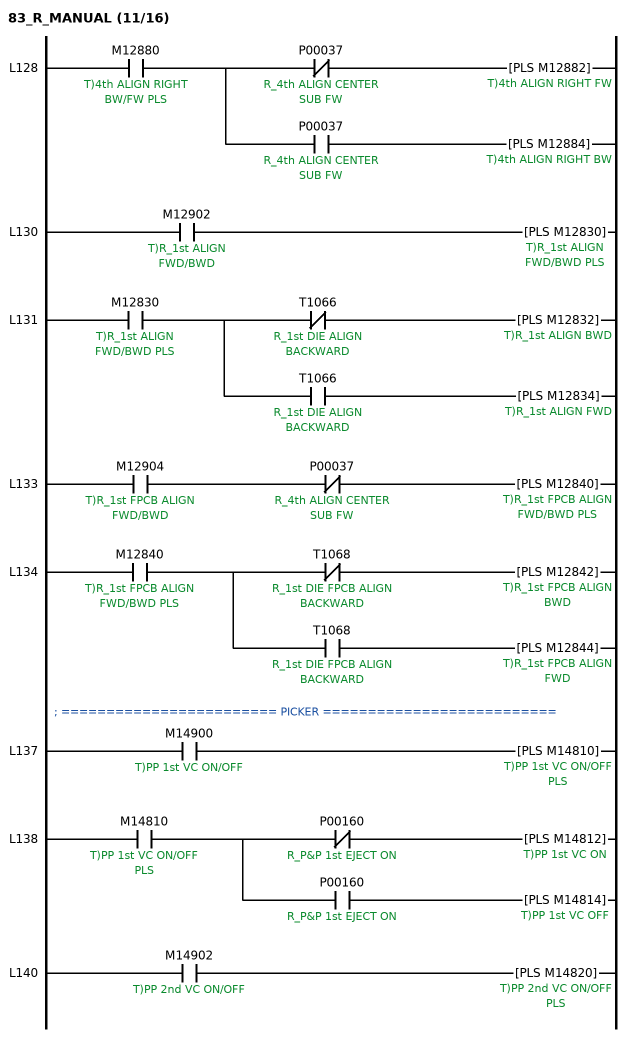
; L128
LOAD      M12880	// T)4th ALIGN RIGHT BW/FW PLS
MPUSH
AND NOT   P00037	// R_4th ALIGN CENTER SUB FW
OUTP      M12882	// T)4th ALIGN RIGHT FW
MPOP
AND       P00037	// R_4th ALIGN CENTER SUB FW
OUTP      M12884	// T)4th ALIGN RIGHT BW
; L130
LOAD      M12902	// T)R_1st ALIGN FWD/BWD
OUTP      M12830	// T)R_1st ALIGN FWD/BWD PLS
; L131
LOAD      M12830	// T)R_1st ALIGN FWD/BWD PLS
MPUSH
AND NOT   T1066	// R_1st DIE ALIGN BACKWARD
OUTP      M12832	// T)R_1st ALIGN BWD
MPOP
AND       T1066	// R_1st DIE ALIGN BACKWARD
OUTP      M12834	// T)R_1st ALIGN FWD
; L133
LOAD      M12904	// T)R_1st FPCB ALIGN FWD/BWD
AND NOT   P00037	// R_4th ALIGN CENTER SUB FW
OUTP      M12840	// T)R_1st FPCB ALIGN FWD/BWD PLS
; L134
LOAD      M12840	// T)R_1st FPCB ALIGN FWD/BWD PLS
MPUSH
AND NOT   T1068	// R_1st DIE FPCB ALIGN BACKWARD
OUTP      M12842	// T)R_1st FPCB ALIGN BWD
MPOP
AND       T1068	// R_1st DIE FPCB ALIGN BACKWARD
OUTP      M12844	// T)R_1st FPCB ALIGN FWD
// ======================== PICKER ==========================
; L137
LOAD      M14900	// T)PP 1st VC ON/OFF
OUTP      M14810	// T)PP 1st VC ON/OFF PLS
; L138
LOAD      M14810	// T)PP 1st VC ON/OFF PLS
MPUSH
AND NOT   P00160	// R_P&P 1st EJECT ON
OUTP      M14812	// T)PP 1st VC ON
MPOP
AND       P00160	// R_P&P 1st EJECT ON
OUTP      M14814	// T)PP 1st VC OFF
; L140
LOAD      M14902	// T)PP 2nd VC ON/OFF
OUTP      M14820	// T)PP 2nd VC ON/OFF PLS

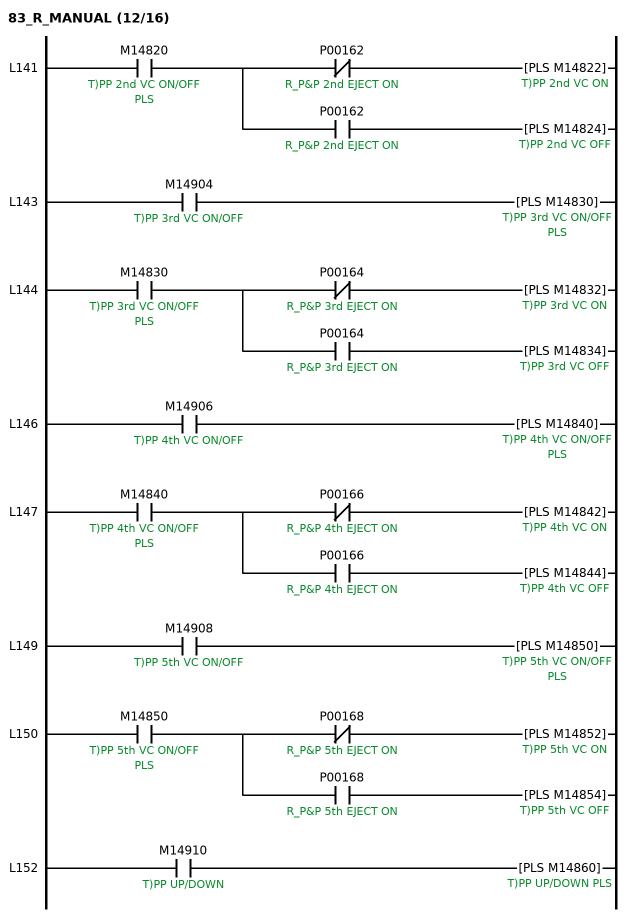
; L141
LOAD      M14820	// T)PP 2nd VC ON/OFF PLS
MPUSH
AND NOT   P00162	// R_P&P 2nd EJECT ON
OUTP      M14822	// T)PP 2nd VC ON
MPOP
AND       P00162	// R_P&P 2nd EJECT ON
OUTP      M14824	// T)PP 2nd VC OFF
; L143
LOAD      M14904	// T)PP 3rd VC ON/OFF
OUTP      M14830	// T)PP 3rd VC ON/OFF PLS
; L144
LOAD      M14830	// T)PP 3rd VC ON/OFF PLS
MPUSH
AND NOT   P00164	// R_P&P 3rd EJECT ON
OUTP      M14832	// T)PP 3rd VC ON
MPOP
AND       P00164	// R_P&P 3rd EJECT ON
OUTP      M14834	// T)PP 3rd VC OFF
; L146
LOAD      M14906	// T)PP 4th VC ON/OFF
OUTP      M14840	// T)PP 4th VC ON/OFF PLS
; L147
LOAD      M14840	// T)PP 4th VC ON/OFF PLS
MPUSH
AND NOT   P00166	// R_P&P 4th EJECT ON
OUTP      M14842	// T)PP 4th VC ON
MPOP
AND       P00166	// R_P&P 4th EJECT ON
OUTP      M14844	// T)PP 4th VC OFF
; L149
LOAD      M14908	// T)PP 5th VC ON/OFF
OUTP      M14850	// T)PP 5th VC ON/OFF PLS
; L150
LOAD      M14850	// T)PP 5th VC ON/OFF PLS
MPUSH
AND NOT   P00168	// R_P&P 5th EJECT ON
OUTP      M14852	// T)PP 5th VC ON
MPOP
AND       P00168	// R_P&P 5th EJECT ON
OUTP      M14854	// T)PP 5th VC OFF
; L152
LOAD      M14910	// T)PP UP/DOWN
OUTP      M14860	// T)PP UP/DOWN PLS

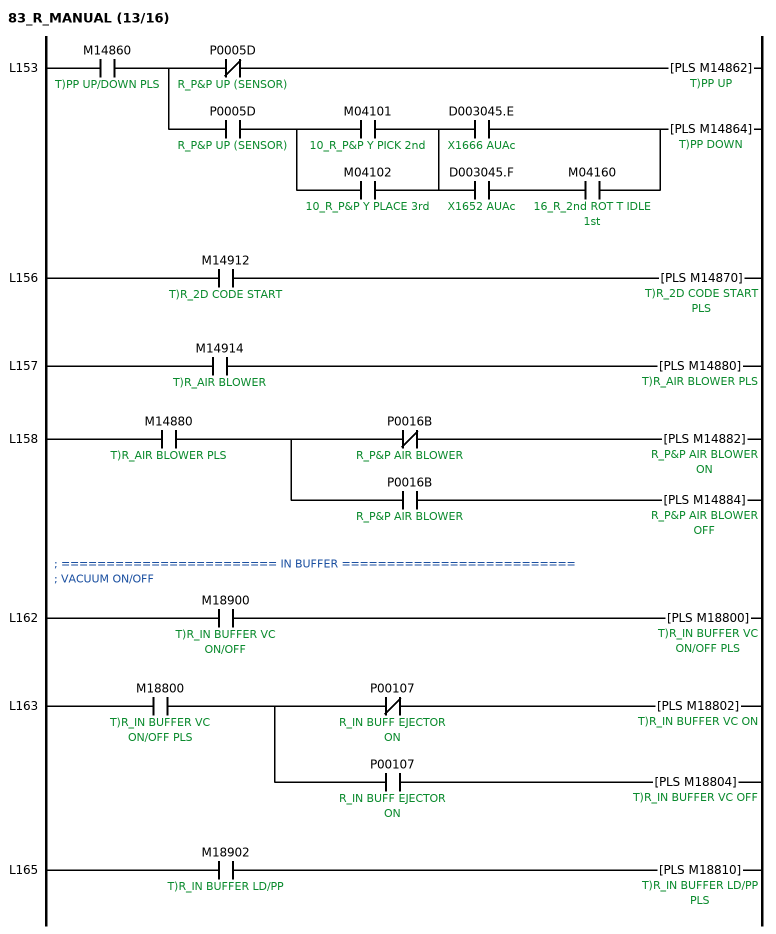
; L153
LOAD      M14860	// T)PP UP/DOWN PLS
MPUSH
AND NOT   P0005D	// R_P&P UP (SENSOR)
OUTP      M14862	// T)PP UP
MPOP
AND       P0005D	// R_P&P UP (SENSOR)
LOAD      M04101	// 10_R_P&P Y PICK 2nd
OR        M04102	// 10_R_P&P Y PLACE 3rd
AND LOAD
LOAD      D003045.E	// X1666 AUAc
LOAD      D003045.F	// X1652 AUAc
AND       M04160	// 16_R_2nd ROT T IDLE 1st
OR LOAD
AND LOAD
OUTP      M14864	// T)PP DOWN
; L156
LOAD      M14912	// T)R_2D CODE START
OUTP      M14870	// T)R_2D CODE START PLS
; L157
LOAD      M14914	// T)R_AIR BLOWER
OUTP      M14880	// T)R_AIR BLOWER PLS
; L158
LOAD      M14880	// T)R_AIR BLOWER PLS
MPUSH
AND NOT   P0016B	// R_P&P AIR BLOWER
OUTP      M14882	// R_P&P AIR BLOWER ON
MPOP
AND       P0016B	// R_P&P AIR BLOWER
OUTP      M14884	// R_P&P AIR BLOWER OFF
// ======================== IN BUFFER ==========================
// VACUUM ON/OFF
; L162
LOAD      M18900	// T)R_IN BUFFER VC ON/OFF
OUTP      M18800	// T)R_IN BUFFER VC ON/OFF PLS
; L163
LOAD      M18800	// T)R_IN BUFFER VC ON/OFF PLS
MPUSH
AND NOT   P00107	// R_IN BUFF EJECTOR ON
OUTP      M18802	// T)R_IN BUFFER VC ON
MPOP
AND       P00107	// R_IN BUFF EJECTOR ON
OUTP      M18804	// T)R_IN BUFFER VC OFF
; L165
LOAD      M18902	// T)R_IN BUFFER LD/PP
OUTP      M18810	// T)R_IN BUFFER LD/PP PLS

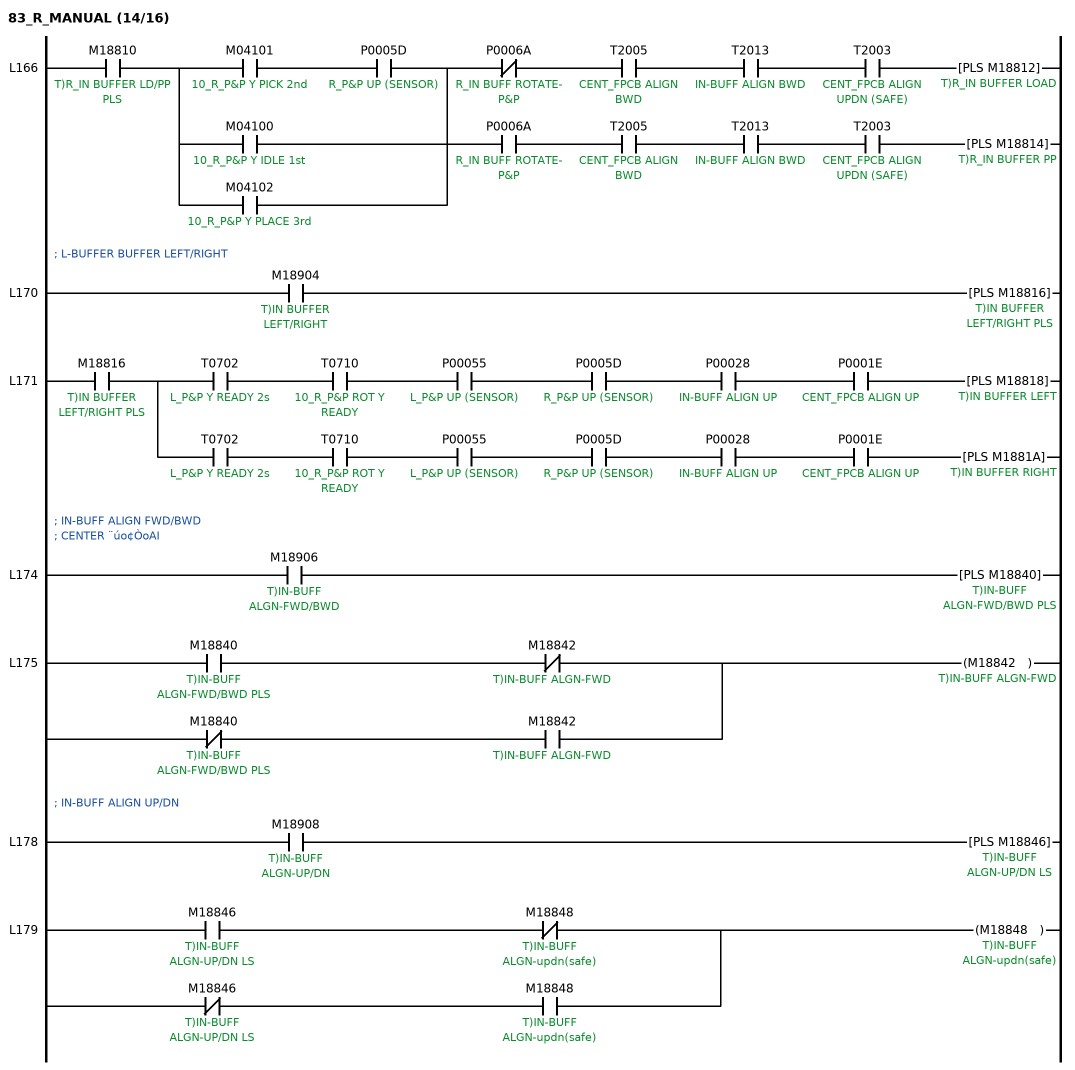
; L166
LOAD      M18810	// T)R_IN BUFFER LD/PP PLS
LOAD      M04101	// 10_R_P&P Y PICK 2nd
AND       P0005D	// R_P&P UP (SENSOR)
OR        M04100	// 10_R_P&P Y IDLE 1st
OR        M04102	// 10_R_P&P Y PLACE 3rd
AND LOAD
MPUSH
AND NOT   P0006A	// R_IN BUFF ROTATE- P&P
AND       T2005	// CENT_FPCB ALIGN BWD
AND       T2013	// IN-BUFF ALIGN BWD
AND       T2003	// CENT_FPCB ALIGN UPDN (SAFE)
OUTP      M18812	// T)R_IN BUFFER LOAD
MPOP
AND       P0006A	// R_IN BUFF ROTATE- P&P
AND       T2005	// CENT_FPCB ALIGN BWD
AND       T2013	// IN-BUFF ALIGN BWD
AND       T2003	// CENT_FPCB ALIGN UPDN (SAFE)
OUTP      M18814	// T)R_IN BUFFER PP
// L-BUFFER BUFFER LEFT/RIGHT
; L170
LOAD      M18904	// T)IN BUFFER LEFT/RIGHT
OUTP      M18816	// T)IN BUFFER LEFT/RIGHT PLS
; L171
LOAD      M18816	// T)IN BUFFER LEFT/RIGHT PLS
MPUSH
AND       T0702	// L_P&P Y READY 2s
AND       T0710	// 10_R_P&P ROT Y READY
AND       P00055	// L_P&P UP (SENSOR)
AND       P0005D	// R_P&P UP (SENSOR)
AND       P00028	// IN-BUFF ALIGN UP
AND       P0001E	// CENT_FPCB ALIGN UP
OUTP      M18818	// T)IN BUFFER LEFT
MPOP
AND       T0702	// L_P&P Y READY 2s
AND       T0710	// 10_R_P&P ROT Y READY
AND       P00055	// L_P&P UP (SENSOR)
AND       P0005D	// R_P&P UP (SENSOR)
AND       P00028	// IN-BUFF ALIGN UP
AND       P0001E	// CENT_FPCB ALIGN UP
OUTP      M1881A	// T)IN BUFFER RIGHT
// IN-BUFF ALIGN FWD/BWD
; L174
LOAD      M18906	// T)IN-BUFF ALGN-FWD/BWD
OUTP      M18840	// T)IN-BUFF ALGN-FWD/BWD PLS
// output comment: CENTER ¨úo¢ÒoAI
; L175
LOAD      M18840	// T)IN-BUFF ALGN-FWD/BWD PLS
AND NOT   M18842	// T)IN-BUFF ALGN-FWD
LOAD NOT  M18840	// T)IN-BUFF ALGN-FWD/BWD PLS
AND       M18842	// T)IN-BUFF ALGN-FWD
OR LOAD
OUT       M18842	// T)IN-BUFF ALGN-FWD
// IN-BUFF ALIGN UP/DN
; L178
LOAD      M18908	// T)IN-BUFF ALGN-UP/DN
OUTP      M18846	// T)IN-BUFF ALGN-UP/DN LS
; L179
LOAD      M18846	// T)IN-BUFF ALGN-UP/DN LS
AND NOT   M18848	// T)IN-BUFF ALGN-updn(safe)
LOAD NOT  M18846	// T)IN-BUFF ALGN-UP/DN LS
AND       M18848	// T)IN-BUFF ALGN-updn(safe)
OR LOAD
OUT       M18848	// T)IN-BUFF ALGN-updn(safe)

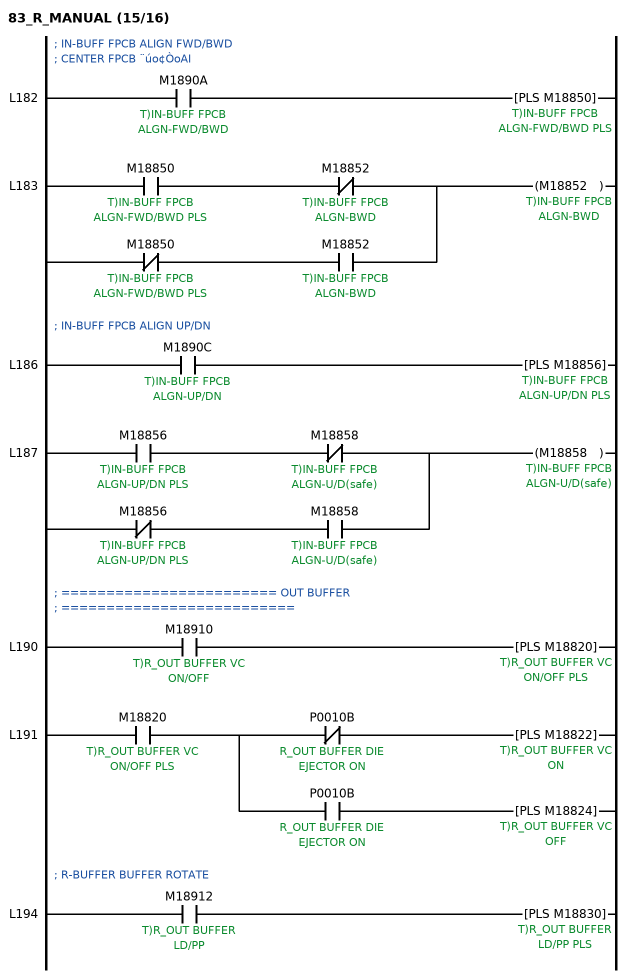
// IN-BUFF FPCB ALIGN FWD/BWD
; L182
LOAD      M1890A	// T)IN-BUFF FPCB ALGN-FWD/BWD
OUTP      M18850	// T)IN-BUFF FPCB ALGN-FWD/BWD PLS
// output comment: CENTER FPCB ¨úo¢ÒoAI
; L183
LOAD      M18850	// T)IN-BUFF FPCB ALGN-FWD/BWD PLS
AND NOT   M18852	// T)IN-BUFF FPCB ALGN-BWD
LOAD NOT  M18850	// T)IN-BUFF FPCB ALGN-FWD/BWD PLS
AND       M18852	// T)IN-BUFF FPCB ALGN-BWD
OR LOAD
OUT       M18852	// T)IN-BUFF FPCB ALGN-BWD
// IN-BUFF FPCB ALIGN UP/DN
; L186
LOAD      M1890C	// T)IN-BUFF FPCB ALGN-UP/DN
OUTP      M18856	// T)IN-BUFF FPCB ALGN-UP/DN PLS
; L187
LOAD      M18856	// T)IN-BUFF FPCB ALGN-UP/DN PLS
AND NOT   M18858	// T)IN-BUFF FPCB ALGN-U/D(safe)
LOAD NOT  M18856	// T)IN-BUFF FPCB ALGN-UP/DN PLS
AND       M18858	// T)IN-BUFF FPCB ALGN-U/D(safe)
OR LOAD
OUT       M18858	// T)IN-BUFF FPCB ALGN-U/D(safe)
// ======================== OUT BUFFER ==========================
; L190
LOAD      M18910	// T)R_OUT BUFFER VC ON/OFF
OUTP      M18820	// T)R_OUT BUFFER VC ON/OFF PLS
; L191
LOAD      M18820	// T)R_OUT BUFFER VC ON/OFF PLS
MPUSH
AND NOT   P0010B	// R_OUT BUFFER DIE EJECTOR ON
OUTP      M18822	// T)R_OUT BUFFER VC ON
MPOP
AND       P0010B	// R_OUT BUFFER DIE EJECTOR ON
OUTP      M18824	// T)R_OUT BUFFER VC OFF
// R-BUFFER BUFFER ROTATE
; L194
LOAD      M18912	// T)R_OUT BUFFER LD/PP
OUTP      M18830	// T)R_OUT BUFFER LD/PP PLS

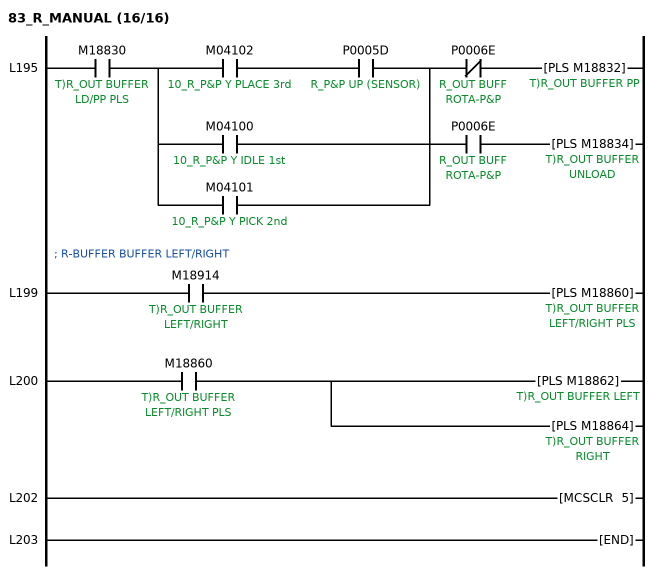
; L195
LOAD      M18830	// T)R_OUT BUFFER LD/PP PLS
LOAD      M04102	// 10_R_P&P Y PLACE 3rd
AND       P0005D	// R_P&P UP (SENSOR)
OR        M04100	// 10_R_P&P Y IDLE 1st
OR        M04101	// 10_R_P&P Y PICK 2nd
AND LOAD
MPUSH
AND NOT   P0006E	// R_OUT BUFF ROTA-P&P
OUTP      M18832	// T)R_OUT BUFFER PP
MPOP
AND       P0006E	// R_OUT BUFF ROTA-P&P
OUTP      M18834	// T)R_OUT BUFFER UNLOAD
// R-BUFFER BUFFER LEFT/RIGHT
; L199
LOAD      M18914	// T)R_OUT BUFFER LEFT/RIGHT
OUTP      M18860	// T)R_OUT BUFFER LEFT/RIGHT PLS
; L200
LOAD      M18860	// T)R_OUT BUFFER LEFT/RIGHT PLS
OUTP      M18862	// T)R_OUT BUFFER LEFT
OUTP      M18864	// T)R_OUT BUFFER RIGHT
; L202
MCSCLR    5
; L203
END

PROGRAM 84_RUN_TIME (task: ¨ö¨¬A¥ì CA¡¤I¡¾¡¿¡¤¡Í)

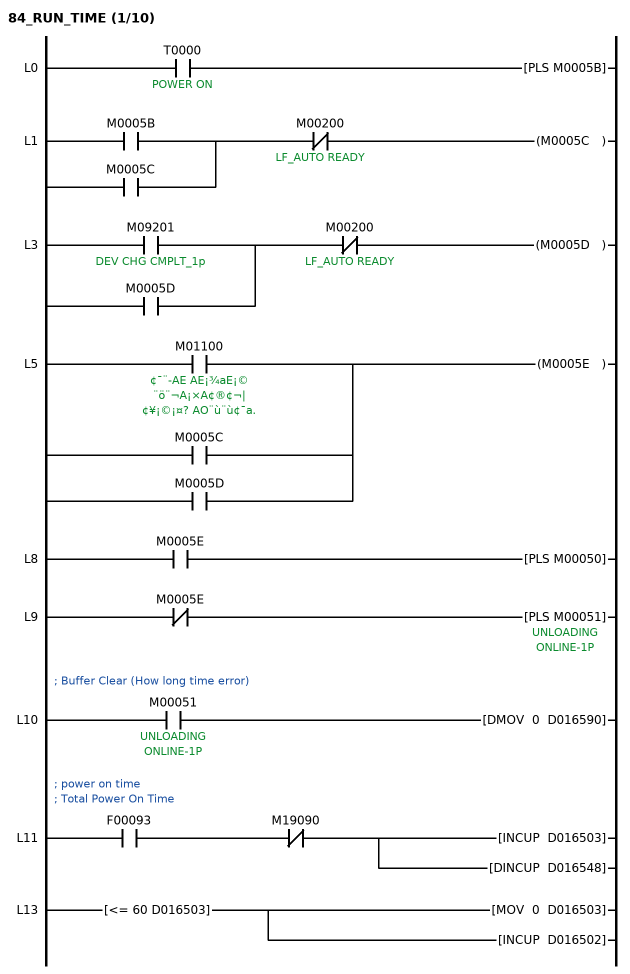
; L0
LOAD      T0000	// POWER ON
OUTP      M0005B
; L1
LOAD      M0005B
OR        M0005C
AND NOT   M00200	// LF_AUTO READY
OUT       M0005C
; L3
LOAD      M09201	// DEV CHG CMPLT_1p
OR        M0005D
AND NOT   M00200	// LF_AUTO READY
OUT       M0005D
; L5
LOAD      M01100	// ¢¯¨­AE AE¡¾aE¡© ¨ö¨¬A¡×A¢®¢¬| ¢¥¡©¡¤? AO¨ù¨ù¢¯a.
OR        M0005C
OR        M0005D
OUT       M0005E
; L8
LOAD      M0005E
OUTP      M00050
; L9
LOAD NOT  M0005E
OUTP      M00051	// UNLOADING ONLINE-1P
; L10
LOAD      M00051	// UNLOADING ONLINE-1P
DMOV      0 D016590
// output comment: Buffer Clear (How long time error)
; L11
LOAD      F00093
AND NOT   M19090
INCUP     D016503
DINCUP    D016548
// output comment: power on time
// output comment: Total Power On Time
; L13
LOAD<=    60 D016503
MOV       0 D016503
INCUP     D016502

